Staubli VAL3: readText.dtx

public bool bBYPASS
public bool bCycle
public bool bCycleEnd = true
bool bGetSpeed = true
bool bMatlab
bool bReadEnd = true
bool bReadWait
public bool bResumeCycle
bool bTxtHeadOk
public bool bWriteEnd = true
frame fPrdFrame = {x=1610.363, y=33.376, z=-220.436, rx=-0.03, ry=0.18, rz=-39.644, fatherId=world[0]}
jointRx jJointRead[100]
  [0] = {j1=8.22, j2=20.1, j3=107.19, j4=-141.77, j5=44.38, j6=150.9}
  [1] = {j1=8.22, j2=20.1, j3=107.19, j4=-141.77, j5=44.38, j6=150.9}
public jointRx jPrdHome = {j1=40.635, j2=24.616, j3=104.715, j4=-108.663, j5=68.526, j6=132.709}
mdesc mNomSpeed = {accel=16, vel=40, decel=16, tmax=80, blend=off, leave=20, reach=20}
public mdesc mSpdOfJnt[100]
  [0] = {accel=40, vel=40, decel=40, rmax=1000, tmax=40, blend=cartesian, leave=0, reach=2}
  [1] = {accel=40, vel=40, decel=40, rmax=1000, tmax=40, blend=cartesian, leave=0, reach=2}
  [2] = {accel=30, vel=40, decel=30, rmax=1000, tmax=15.702, blend=cartesian, leave=0, reach=2}
  [3] = {accel=30, vel=40, decel=30, rmax=1000, tmax=6.112, blend=cartesian, leave=0, reach=2}
  [4] = {accel=16, vel=40, decel=16, rmax=1000, tmax=200, blend=cartesian, leave=2, reach=2}
  [5] = {accel=16, vel=40, decel=16, rmax=1000, tmax=200, blend=cartesian, leave=2, reach=2}
  [6] = {accel=16, vel=40, decel=16, rmax=1000, tmax=200, blend=cartesian, leave=2, reach=2}
  [7] = {accel=16, vel=40, decel=16, rmax=1000, tmax=200, blend=cartesian, leave=2, reach=2}
  [8] = {accel=16, vel=40, decel=16, rmax=1000, tmax=200, blend=cartesian, leave=2, reach=2}
  [9] = {accel=16, vel=40, decel=16, rmax=1000, tmax=200, blend=cartesian, leave=2, reach=2}
  [10] = {accel=16, vel=40, decel=16, rmax=1000, tmax=200, blend=cartesian, leave=2, reach=2}
  [11] = {accel=16, vel=40, decel=16, rmax=1000, tmax=200, blend=cartesian, leave=2, reach=2}
  [12] = {accel=16, vel=40, decel=16, rmax=1000, tmax=200, blend=cartesian, leave=2, reach=2}
  [13] = {accel=16, vel=40, decel=16, rmax=1000, tmax=200, blend=cartesian, leave=2, reach=2}
  [14] = {accel=16, vel=40, decel=16, rmax=1000, tmax=200, blend=cartesian, leave=2, reach=2}
  [15] = {accel=16, vel=40, decel=16, rmax=1000, tmax=200, blend=cartesian, leave=2, reach=2}
  [16] = {accel=16, vel=40, decel=16, rmax=1000, tmax=200, blend=cartesian, leave=2, reach=2}
  [17] = {accel=16, vel=40, decel=16, rmax=1000, tmax=200, blend=cartesian, leave=2, reach=2}
  [18] = {accel=16, vel=40, decel=16, rmax=1000, tmax=200, blend=cartesian, leave=2, reach=2}
  [19] = {accel=16, vel=40, decel=16, rmax=1000, tmax=200, blend=cartesian, leave=2, reach=2}
  [20] = {accel=16, vel=40, decel=16, rmax=1000, tmax=200, blend=cartesian, leave=2, reach=2}
  [21] = {accel=16, vel=40, decel=16, rmax=1000, tmax=200, blend=cartesian, leave=2, reach=2}
  [22] = {accel=16, vel=40, decel=16, rmax=1000, tmax=200, blend=cartesian, leave=2, reach=2}
  [23] = {accel=16, vel=40, decel=16, rmax=1000, tmax=200, blend=cartesian, leave=2, reach=2}
  [24] = {accel=16, vel=40, decel=16, rmax=1000, tmax=200, blend=cartesian, leave=2, reach=2}
  [25] = {accel=16, vel=40, decel=16, rmax=1000, tmax=200, blend=cartesian, leave=2, reach=2}
  [26] = {accel=16, vel=40, decel=16, rmax=1000, tmax=200, blend=cartesian, leave=2, reach=2}
  [27] = {accel=16, vel=40, decel=16, rmax=1000, tmax=200, blend=cartesian, leave=2, reach=2}
  [28] = {accel=16, vel=40, decel=16, rmax=1000, tmax=200, blend=cartesian, leave=2, reach=2}
  [29] = {accel=16, vel=40, decel=16, rmax=1000, tmax=200, blend=cartesian, leave=2, reach=2}
  [30] = {accel=16, vel=40, decel=16, rmax=1000, tmax=200, blend=cartesian, leave=2, reach=2}
  [31] = {accel=16, vel=40, decel=16, rmax=1000, tmax=200, blend=cartesian, leave=2, reach=2}
  [32] = {accel=16, vel=40, decel=16, rmax=1000, tmax=200, blend=cartesian, leave=2, reach=2}
  [33] = {accel=16, vel=40, decel=16, rmax=1000, tmax=200, blend=cartesian, leave=2, reach=2}
  [34] = {accel=16, vel=40, decel=16, rmax=1000, tmax=200, blend=cartesian, leave=2, reach=2}
  [35] = {accel=16, vel=40, decel=16, rmax=1000, tmax=200, blend=cartesian, leave=2, reach=2}
  [36] = {accel=16, vel=40, decel=16, rmax=1000, tmax=200, blend=cartesian, leave=2, reach=2}
  [37] = {accel=16, vel=40, decel=16, rmax=1000, tmax=200, blend=cartesian, leave=2, reach=2}
  [38] = {accel=16, vel=40, decel=16, rmax=1000, tmax=200, blend=cartesian, leave=2, reach=2}
  [39] = {accel=16, vel=40, decel=16, rmax=1000, tmax=200, blend=cartesian, leave=2, reach=2}
  [40] = {accel=16, vel=40, decel=16, rmax=1000, tmax=200, blend=cartesian, leave=2, reach=2}
  [41] = {accel=16, vel=40, decel=16, rmax=1000, tmax=200, blend=cartesian, leave=2, reach=2}
  [42] = {accel=16, vel=40, decel=16, rmax=1000, tmax=200, blend=cartesian, leave=2, reach=2}
  [43] = {accel=16, vel=40, decel=16, rmax=1000, tmax=200, blend=cartesian, leave=2, reach=2}
  [44] = {accel=16, vel=40, decel=16, rmax=1000, tmax=200, blend=cartesian, leave=2, reach=2}
  [45] = {accel=16, vel=40, decel=16, rmax=1000, tmax=200, blend=cartesian, leave=2, reach=2}
  [46] = {accel=16, vel=40, decel=16, rmax=1000, tmax=200, blend=cartesian, leave=2, reach=2}
  [47] = {accel=16, vel=40, decel=16, rmax=1000, tmax=200, blend=cartesian, leave=2, reach=2}
  [48] = {accel=16, vel=40, decel=16, rmax=1000, tmax=200, blend=cartesian, leave=2, reach=2}
  [49] = {accel=16, vel=40, decel=16, rmax=1000, tmax=200, blend=cartesian, leave=2, reach=2}
  [50] = {accel=16, vel=40, decel=16, rmax=1000, tmax=200, blend=cartesian, leave=2, reach=2}
  [51] = {accel=16, vel=40, decel=16, rmax=1000, tmax=200, blend=cartesian, leave=2, reach=2}
  [52] = {accel=16, vel=40, decel=16, rmax=1000, tmax=200, blend=cartesian, leave=2, reach=2}
  [53] = {accel=16, vel=40, decel=16, rmax=1000, tmax=200, blend=cartesian, leave=2, reach=2}
  [54] = {accel=16, vel=40, decel=16, rmax=1000, tmax=200, blend=cartesian, leave=2, reach=2}
  [55] = {accel=16, vel=40, decel=16, rmax=1000, tmax=200, blend=cartesian, leave=2, reach=2}
  [56] = {accel=16, vel=40, decel=16, rmax=1000, tmax=200, blend=cartesian, leave=2, reach=2}
  [57] = {accel=16, vel=40, decel=16, rmax=1000, tmax=200, blend=cartesian, leave=2, reach=2}
  [58] = {accel=16, vel=40, decel=16, rmax=1000, tmax=200, blend=cartesian, leave=2, reach=2}
  [59] = {accel=16, vel=40, decel=16, rmax=1000, tmax=200, blend=cartesian, leave=2, reach=2}
  [60] = {accel=16, vel=40, decel=16, rmax=1000, tmax=200, blend=cartesian, leave=2, reach=2}
  [61] = {accel=16, vel=40, decel=16, rmax=1000, tmax=200, blend=cartesian, leave=2, reach=2}
  [62] = {accel=16, vel=40, decel=16, rmax=1000, tmax=200, blend=cartesian, leave=2, reach=2}
  [63] = {accel=16, vel=40, decel=16, rmax=1000, tmax=200, blend=cartesian, leave=2, reach=2}
  [64] = {accel=16, vel=40, decel=16, rmax=1000, tmax=200, blend=cartesian, leave=2, reach=2}
  [65] = {accel=16, vel=40, decel=16, rmax=1000, tmax=200, blend=cartesian, leave=2, reach=2}
  [66] = {accel=16, vel=40, decel=16, rmax=1000, tmax=200, blend=cartesian, leave=2, reach=2}
  [67] = {accel=16, vel=40, decel=16, rmax=1000, tmax=200, blend=cartesian, leave=2, reach=2}
  [68] = {accel=16, vel=40, decel=16, rmax=1000, tmax=200, blend=cartesian, leave=2, reach=2}
  [69] = {accel=16, vel=40, decel=16, rmax=1000, tmax=200, blend=cartesian, leave=2, reach=2}
  [70] = {accel=16, vel=40, decel=16, rmax=1000, tmax=200, blend=cartesian, leave=2, reach=2}
  [71] = {accel=16, vel=40, decel=16, rmax=1000, tmax=200, blend=cartesian, leave=2, reach=2}
  [72] = {accel=16, vel=40, decel=16, rmax=1000, tmax=200, blend=cartesian, leave=2, reach=2}
  [73] = {accel=16, vel=40, decel=16, rmax=1000, tmax=200, blend=cartesian, leave=2, reach=2}
  [74] = {accel=16, vel=40, decel=16, rmax=1000, tmax=200, blend=cartesian, leave=2, reach=2}
  [75] = {accel=16, vel=40, decel=16, rmax=1000, tmax=200, blend=cartesian, leave=2, reach=2}
  [76] = {accel=16, vel=40, decel=16, rmax=1000, tmax=200, blend=cartesian, leave=2, reach=2}
  [77] = {accel=16, vel=40, decel=16, rmax=1000, tmax=200, blend=cartesian, leave=2, reach=2}
  [78] = {accel=16, vel=40, decel=16, rmax=1000, tmax=200, blend=cartesian, leave=2, reach=2}
  [79] = {accel=16, vel=40, decel=16, rmax=1000, tmax=200, blend=cartesian, leave=2, reach=2}
  [80] = {accel=16, vel=40, decel=16, rmax=1000, tmax=200, blend=cartesian, leave=2, reach=2}
  [81] = {accel=16, vel=40, decel=16, rmax=1000, tmax=200, blend=cartesian, leave=2, reach=2}
  [82] = {accel=16, vel=40, decel=16, rmax=1000, tmax=200, blend=cartesian, leave=2, reach=2}
  [83] = {accel=16, vel=40, decel=16, rmax=1000, tmax=200, blend=cartesian, leave=2, reach=2}
  [84] = {accel=16, vel=40, decel=16, rmax=1000, tmax=200, blend=cartesian, leave=2, reach=2}
  [85] = {accel=16, vel=40, decel=16, rmax=1000, tmax=200, blend=cartesian, leave=2, reach=2}
  [86] = {accel=16, vel=40, decel=16, rmax=1000, tmax=200, blend=cartesian, leave=2, reach=2}
  [87] = {accel=16, vel=40, decel=16, rmax=1000, tmax=200, blend=cartesian, leave=2, reach=2}
  [88] = {accel=16, vel=40, decel=16, rmax=1000, tmax=200, blend=cartesian, leave=2, reach=2}
  [89] = {accel=16, vel=40, decel=16, rmax=1000, tmax=200, blend=cartesian, leave=2, reach=2}
  [90] = {accel=16, vel=40, decel=16, rmax=1000, tmax=200, blend=cartesian, leave=2, reach=2}
  [91] = {accel=16, vel=40, decel=16, rmax=1000, tmax=200, blend=cartesian, leave=2, reach=2}
  [92] = {accel=16, vel=40, decel=16, rmax=1000, tmax=200, blend=cartesian, leave=2, reach=2}
  [93] = {accel=16, vel=40, decel=16, rmax=1000, tmax=200, blend=cartesian, leave=2, reach=2}
  [94] = {accel=16, vel=40, decel=16, rmax=1000, tmax=200, blend=cartesian, leave=2, reach=2}
  [95] = {accel=16, vel=40, decel=16, rmax=1000, tmax=200, blend=cartesian, leave=2, reach=2}
  [96] = {accel=16, vel=40, decel=16, rmax=1000, tmax=200, blend=cartesian, leave=2, reach=2}
  [97] = {accel=16, vel=40, decel=16, rmax=1000, tmax=200, blend=cartesian, leave=2, reach=2}
  [98] = {accel=16, vel=40, decel=16, rmax=1000, tmax=200, blend=cartesian, leave=2, reach=2}
  [99] = {accel=16, vel=40, decel=16, rmax=1000, tmax=200, blend=cartesian, leave=2, reach=2}
public mdesc mSpdOfPt[1000]
  [0] = {accel=80, decel=80, tmax=12.678, leave=0.5, reach=0.5}
  [1] = {accel=80, decel=80, tmax=11.985, leave=0.5, reach=0.5}
  [2] = {accel=80, decel=80, tmax=11.817, leave=0.5, reach=0.5}
  [3] = {accel=80, decel=80, tmax=11.196, leave=0.5, reach=0.5}
  [4] = {accel=80, decel=80, tmax=9.277, leave=0.5, reach=0.5}
  [5] = {accel=80, decel=80, tmax=7.453, leave=0.5, reach=0.5}
  [6] = {accel=80, decel=80, tmax=6.952, leave=0.5, reach=0.5}
  [7] = {accel=80, decel=80, tmax=7.802, leave=0.5, reach=0.5}
  [8] = {accel=80, decel=80, tmax=10.02, leave=0.5, reach=0.5}
  [9] = {accel=80, decel=80, tmax=12.345, leave=0.5, reach=0.5}
  [10] = {accel=80, decel=80, tmax=14.425, leave=0.5, reach=0.5}
  [11] = {accel=80, decel=80, tmax=15.256, leave=0.5, reach=0.5}
  [12] = {accel=80, decel=80, tmax=15.163, leave=0.5, reach=0.5}
  [13] = {accel=80, decel=80, tmax=13.825, leave=0.5, reach=0.5}
  [14] = {accel=80, decel=80, tmax=12.953, leave=0.5, reach=0.5}
  [15] = {accel=80, decel=80, tmax=11.37, leave=0.5, reach=0.5}
  [16] = {accel=80, decel=80, tmax=9.559, leave=0.5, reach=0.5}
  [17] = {accel=80, decel=80, tmax=9.004, leave=0.5, reach=0.5}
  [18] = {accel=80, decel=80, tmax=10.189, leave=0.5, reach=0.5}
  [19] = {accel=80, decel=80, tmax=12.733, leave=0.5, reach=0.5}
  [20] = {accel=80, decel=80, tmax=10.204, leave=0.5, reach=0.5}
  [21] = {accel=80, decel=80, tmax=6.338, leave=0.5, reach=0.5}
  [22] = {accel=80, decel=80, tmax=4.399, leave=0.5, reach=0.5}
  [23] = {accel=80, decel=80, tmax=3.23, leave=0.5, reach=0.5}
  [24] = {accel=80, decel=80, tmax=3.6, leave=0.5, reach=0.5}
  [25] = {accel=80, decel=80, tmax=5.733, leave=0.5, reach=0.5}
  [26] = {accel=80, decel=80, tmax=10.337, leave=0.5, reach=0.5}
  [27] = {accel=80, decel=80, tmax=12.442, leave=0.5, reach=0.5}
  [28] = {accel=80, decel=80, tmax=8.009, leave=0.5, reach=0.5}
  [29] = {accel=80, decel=80, tmax=7.489, leave=0.5, reach=0.5}
  [30] = {accel=80, decel=80, tmax=9.024, leave=0.5, reach=0.5}
  [31] = {accel=80, decel=80, tmax=10.72, leave=0.5, reach=0.5}
  [32] = {accel=80, decel=80, tmax=13.479, leave=0.5, reach=0.5}
  [33] = {accel=80, decel=80, tmax=15.007, leave=0.5, reach=0.5}
  [34] = {accel=80, decel=80, tmax=16.256, leave=0.5, reach=0.5}
  [35] = {accel=80, decel=80, tmax=14.52, leave=0.5, reach=0.5}
  [36] = {accel=80, decel=80, tmax=13.789, leave=0.5, reach=0.5}
  [37] = {accel=80, decel=80, tmax=13.032, leave=0.5, reach=0.5}
  [38] = {accel=80, decel=80, tmax=10.441, leave=0.5, reach=0.5}
  [39] = {accel=80, decel=80, tmax=8.528, leave=0.5, reach=0.5}
  [40] = {accel=80, decel=80, tmax=7.32, leave=0.5, reach=0.5}
  [41] = {accel=80, decel=80, tmax=7.727, leave=0.5, reach=0.5}
  [42] = {accel=80, decel=80, tmax=9.914, leave=0.5, reach=0.5}
  [43] = {accel=80, decel=80, tmax=12.183, leave=0.5, reach=0.5}
  [44] = {accel=80, decel=80, tmax=11.946, leave=0.5, reach=0.5}
  [45] = {accel=80, decel=80, tmax=11.661, leave=0.5, reach=0.5}
  [46] = {accel=80, decel=80, tmax=12.164, leave=0.5, reach=0.5}
  [47] = {accel=80, decel=80, tmax=13.305, leave=0.5, reach=0.5}
  [48] = {accel=80, decel=80, tmax=14.537, leave=0.5, reach=0.5}
  [49] = {accel=80, decel=80, tmax=14.655, leave=0.5, reach=0.5}
  [50] = {accel=80, decel=80, tmax=13.906, leave=0.5, reach=0.5}
  [51] = {accel=80, decel=80, tmax=12.405, leave=0.5, reach=0.5}
  [52] = {accel=80, decel=80, tmax=11.068, leave=0.5, reach=0.5}
  [53] = {accel=80, decel=80, tmax=9.816, leave=0.5, reach=0.5}
  [54] = {accel=80, decel=80, tmax=8.99, leave=0.5, reach=0.5}
  [55] = {accel=80, decel=80, tmax=8.736, leave=0.5, reach=0.5}
  [56] = {accel=80, decel=80, tmax=8.829, leave=0.5, reach=0.5}
  [57] = {accel=80, decel=80, tmax=9.678, leave=0.5, reach=0.5}
  [58] = {accel=80, decel=80, tmax=11.32, leave=0.5, reach=0.5}
  [59] = {accel=80, decel=80, tmax=13.047, leave=0.5, reach=0.5}
  [60] = {accel=80, decel=80, tmax=14.414, leave=0.5, reach=0.5}
  [61] = {accel=80, decel=80, tmax=14.8, leave=0.5, reach=0.5}
  [62] = {accel=80, decel=80, tmax=15.263, leave=0.5, reach=0.5}
  [63] = {accel=80, decel=80, tmax=15.263, leave=0.5, reach=0.5}
  [64] = {accel=80, decel=80, tmax=14.8, leave=0.5, reach=0.5}
  [65] = {accel=80, decel=80, tmax=14.414, leave=0.5, reach=0.5}
  [66] = {accel=80, decel=80, tmax=13.047, leave=0.5, reach=0.5}
  [67] = {accel=80, decel=80, tmax=11.32, leave=0.5, reach=0.5}
  [68] = {accel=80, decel=80, tmax=9.678, leave=0.5, reach=0.5}
  [69] = {accel=80, decel=80, tmax=8.829, leave=0.5, reach=0.5}
  [70] = {accel=80, decel=80, tmax=8.736, leave=0.5, reach=0.5}
  [71] = {accel=80, decel=80, tmax=8.99, leave=0.5, reach=0.5}
  [72] = {accel=80, decel=80, tmax=9.816, leave=0.5, reach=0.5}
  [73] = {accel=80, decel=80, tmax=11.068, leave=0.5, reach=0.5}
  [74] = {accel=80, decel=80, tmax=12.405, leave=0.5, reach=0.5}
  [75] = {accel=80, decel=80, tmax=13.906, leave=0.5, reach=0.5}
  [76] = {accel=80, decel=80, tmax=14.655, leave=0.5, reach=0.5}
  [77] = {accel=80, decel=80, tmax=14.537, leave=0.5, reach=0.5}
  [78] = {accel=80, decel=80, tmax=13.305, leave=0.5, reach=0.5}
  [79] = {accel=80, decel=80, tmax=12.164, leave=0.5, reach=0.5}
  [80] = {accel=80, decel=80, tmax=11.661, leave=0.5, reach=0.5}
  [81] = {accel=80, decel=80, tmax=11.946, leave=0.5, reach=0.5}
  [82] = {accel=80, decel=80, tmax=12.183, leave=0.5, reach=0.5}
  [83] = {accel=80, decel=80, tmax=9.914, leave=0.5, reach=0.5}
  [84] = {accel=80, decel=80, tmax=7.727, leave=0.5, reach=0.5}
  [85] = {accel=80, decel=80, tmax=7.32, leave=0.5, reach=0.5}
  [86] = {accel=80, decel=80, tmax=8.528, leave=0.5, reach=0.5}
  [87] = {accel=80, decel=80, tmax=10.441, leave=0.5, reach=0.5}
  [88] = {accel=80, decel=80, tmax=13.032, leave=0.5, reach=0.5}
  [89] = {accel=80, decel=80, tmax=13.789, leave=0.5, reach=0.5}
  [90] = {accel=80, decel=80, tmax=14.52, leave=0.5, reach=0.5}
  [91] = {accel=80, decel=80, tmax=16.256, leave=0.5, reach=0.5}
  [92] = {accel=80, decel=80, tmax=15.007, leave=0.5, reach=0.5}
  [93] = {accel=80, decel=80, tmax=13.479, leave=0.5, reach=0.5}
  [94] = {accel=80, decel=80, tmax=10.72, leave=0.5, reach=0.5}
  [95] = {accel=80, decel=80, tmax=9.024, leave=0.5, reach=0.5}
  [96] = {accel=80, decel=80, tmax=7.489, leave=0.5, reach=0.5}
  [97] = {accel=80, decel=80, tmax=8.009, leave=0.5, reach=0.5}
  [98] = {accel=80, decel=80, tmax=12.442, leave=0.5, reach=0.5}
  [99] = {accel=80, decel=80, tmax=10.337, leave=0.5, reach=0.5}
  [100] = {accel=80, decel=80, tmax=5.733, leave=0.5, reach=0.5}
  [101] = {accel=80, decel=80, tmax=3.6, leave=0.5, reach=0.5}
  [102] = {accel=80, decel=80, tmax=2.543, leave=0.5, reach=0.5}
  [103] = {accel=80, decel=80, tmax=3.382, leave=0.5, reach=0.5}
  [104] = {accel=80, decel=80, tmax=8.429, leave=0.5, reach=0.5}
  [105] = {accel=80, decel=80, tmax=19.886, leave=0.5, reach=0.5}
  [106] = {accel=80, decel=80, tmax=17.791, leave=0.5, reach=0.5}
  [107] = {accel=80, decel=80, tmax=11.419, leave=0.5, reach=0.5}
  [108] = {accel=80, decel=80, tmax=11.37, leave=0.5, reach=0.5}
  [109] = {accel=80, decel=80, tmax=11.627, leave=0.5, reach=0.5}
  [110] = {accel=80, decel=80, tmax=12.894, leave=0.5, reach=0.5}
  [111] = {accel=80, decel=80, tmax=13.668, leave=0.5, reach=0.5}
  [112] = {accel=80, decel=80, tmax=13.576, leave=0.5, reach=0.5}
  [113] = {accel=80, decel=80, tmax=14.175, leave=0.5, reach=0.5}
  [114] = {accel=80, decel=80, tmax=14.134, leave=0.5, reach=0.5}
  [115] = {accel=80, decel=80, tmax=13.985, leave=0.5, reach=0.5}
  [116] = {accel=80, decel=80, tmax=12.607, leave=0.5, reach=0.5}
  [117] = {accel=80, decel=80, tmax=11.516, leave=0.5, reach=0.5}
  [118] = {accel=80, decel=80, tmax=9.221, leave=0.5, reach=0.5}
  [119] = {accel=80, decel=80, tmax=7.688, leave=0.5, reach=0.5}
  [120] = {accel=80, decel=80, tmax=8.33, leave=0.5, reach=0.5}
  [121] = {accel=80, decel=80, tmax=12.323, leave=0.5, reach=0.5}
  [122] = {accel=80, decel=80, tmax=16.24, leave=0.5, reach=0.5}
  [123] = {accel=80, decel=80, tmax=16.452, leave=0.5, reach=0.5}
  [124] = {accel=80, decel=80, tmax=15.039, leave=0.5, reach=0.5}
  [125] = {accel=80, decel=80, tmax=15.151, leave=0.5, reach=0.5}
  [126] = {accel=80, decel=80, tmax=16.662, leave=0.5, reach=0.5}
  [127] = {accel=80, decel=80, tmax=17.112, leave=0.5, reach=0.5}
  [128] = {accel=80, decel=80, tmax=17.817, leave=0.5, reach=0.5}
  [129] = {accel=80, decel=80, tmax=16.855, leave=0.5, reach=0.5}
  [130] = {accel=80, decel=80, tmax=16.144, leave=0.5, reach=0.5}
  [131] = {accel=80, decel=80, tmax=13.939, leave=0.5, reach=0.5}
  [132] = {accel=80, decel=80, tmax=12.086, leave=0.5, reach=0.5}
  [133] = {accel=80, decel=80, tmax=11.201, leave=0.5, reach=0.5}
  [134] = {accel=80, decel=80, tmax=10.554, leave=0.5, reach=0.5}
  [135] = {accel=80, decel=80, tmax=10.969, leave=0.5, reach=0.5}
  [136] = {accel=80, decel=80, tmax=12.181, leave=0.5, reach=0.5}
  [137] = {accel=80, decel=80, tmax=14.738, leave=0.5, reach=0.5}
  [138] = {accel=80, decel=80, tmax=18.232, leave=0.5, reach=0.5}
  [139] = {accel=80, decel=80, tmax=21.108, leave=0.5, reach=0.5}
  [140] = {accel=80, decel=80, tmax=21.399, leave=0.5, reach=0.5}
  [141] = {accel=80, decel=80, tmax=21.285, leave=0.5, reach=0.5}
  [142] = {accel=80, decel=80, tmax=21.285, leave=0.5, reach=0.5}
  [143] = {accel=80, decel=80, tmax=21.399, leave=0.5, reach=0.5}
  [144] = {accel=80, decel=80, tmax=21.108, leave=0.5, reach=0.5}
  [145] = {accel=80, decel=80, tmax=18.232, leave=0.5, reach=0.5}
  [146] = {accel=80, decel=80, tmax=14.738, leave=0.5, reach=0.5}
  [147] = {accel=80, decel=80, tmax=12.181, leave=0.5, reach=0.5}
  [148] = {accel=80, decel=80, tmax=10.969, leave=0.5, reach=0.5}
  [149] = {accel=80, decel=80, tmax=10.554, leave=0.5, reach=0.5}
  [150] = {accel=80, decel=80, tmax=11.201, leave=0.5, reach=0.5}
  [151] = {accel=80, decel=80, tmax=12.086, leave=0.5, reach=0.5}
  [152] = {accel=80, decel=80, tmax=13.939, leave=0.5, reach=0.5}
  [153] = {accel=80, decel=80, tmax=16.144, leave=0.5, reach=0.5}
  [154] = {accel=80, decel=80, tmax=16.855, leave=0.5, reach=0.5}
  [155] = {accel=80, decel=80, tmax=17.817, leave=0.5, reach=0.5}
  [156] = {accel=80, decel=80, tmax=17.112, leave=0.5, reach=0.5}
  [157] = {accel=80, decel=80, tmax=16.662, leave=0.5, reach=0.5}
  [158] = {accel=80, decel=80, tmax=15.151, leave=0.5, reach=0.5}
  [159] = {accel=80, decel=80, tmax=15.039, leave=0.5, reach=0.5}
  [160] = {accel=80, decel=80, tmax=16.452, leave=0.5, reach=0.5}
  [161] = {accel=80, decel=80, tmax=16.24, leave=0.5, reach=0.5}
  [162] = {accel=80, decel=80, tmax=12.323, leave=0.5, reach=0.5}
  [163] = {accel=80, decel=80, tmax=8.33, leave=0.5, reach=0.5}
  [164] = {accel=80, decel=80, tmax=7.688, leave=0.5, reach=0.5}
  [165] = {accel=80, decel=80, tmax=9.221, leave=0.5, reach=0.5}
  [166] = {accel=80, decel=80, tmax=11.516, leave=0.5, reach=0.5}
  [167] = {accel=80, decel=80, tmax=12.607, leave=0.5, reach=0.5}
  [168] = {accel=80, decel=80, tmax=13.985, leave=0.5, reach=0.5}
  [169] = {accel=80, decel=80, tmax=14.134, leave=0.5, reach=0.5}
  [170] = {accel=80, decel=80, tmax=14.175, leave=0.5, reach=0.5}
  [171] = {accel=80, decel=80, tmax=13.576, leave=0.5, reach=0.5}
  [172] = {accel=80, decel=80, tmax=13.668, leave=0.5, reach=0.5}
  [173] = {accel=80, decel=80, tmax=12.894, leave=0.5, reach=0.5}
  [174] = {accel=80, decel=80, tmax=11.627, leave=0.5, reach=0.5}
  [175] = {accel=80, decel=80, tmax=11.37, leave=0.5, reach=0.5}
  [176] = {accel=80, decel=80, tmax=11.419, leave=0.5, reach=0.5}
  [177] = {accel=80, decel=80, tmax=17.791, leave=0.5, reach=0.5}
  [178] = {accel=80, decel=80, tmax=19.886, leave=0.5, reach=0.5}
  [179] = {accel=80, decel=80, tmax=8.429, leave=0.5, reach=0.5}
  [180] = {accel=80, decel=80, tmax=3.382, leave=0.5, reach=0.5}
  [181] = {accel=80, decel=80, tmax=2.528, leave=0.5, reach=0.5}
  [182] = {accel=80, decel=80, tmax=5.122, leave=0.5, reach=0.5}
  [183] = {accel=80, decel=80, tmax=27.24, leave=0.5, reach=0.5}
  [184] = {accel=80, decel=80, tmax=39.096, leave=0.5, reach=0.5}
  [185] = {accel=80, decel=80, tmax=33.981, leave=0.5, reach=0.5}
  [186] = {accel=80, decel=80, tmax=21.665, leave=0.5, reach=0.5}
  [187] = {accel=80, decel=80, tmax=15.615, leave=0.5, reach=0.5}
  [188] = {accel=80, decel=80, tmax=14.794, leave=0.5, reach=0.5}
  [189] = {accel=80, decel=80, tmax=14.111, leave=0.5, reach=0.5}
  [190] = {accel=80, decel=80, tmax=11.648, leave=0.5, reach=0.5}
  [191] = {accel=80, decel=80, tmax=10.193, leave=0.5, reach=0.5}
  [192] = {accel=80, decel=80, tmax=9.944, leave=0.5, reach=0.5}
  [193] = {accel=80, decel=80, tmax=9.415, leave=0.5, reach=0.5}
  [194] = {accel=80, decel=80, tmax=9.98, leave=0.5, reach=0.5}
  [195] = {accel=80, decel=80, tmax=10.948, leave=0.5, reach=0.5}
  [196] = {accel=80, decel=80, tmax=10.247, leave=0.5, reach=0.5}
  [197] = {accel=80, decel=80, tmax=9.066, leave=0.5, reach=0.5}
  [198] = {accel=80, decel=80, tmax=8.169, leave=0.5, reach=0.5}
  [199] = {accel=80, decel=80, tmax=9.444, leave=0.5, reach=0.5}
  [200] = {accel=80, decel=80, tmax=14.904, leave=0.5, reach=0.5}
  [201] = {accel=80, decel=80, tmax=23.746, leave=0.5, reach=0.5}
  [202] = {accel=80, decel=80, tmax=21.93, leave=0.5, reach=0.5}
  [203] = {accel=80, decel=80, tmax=18.32, leave=0.5, reach=0.5}
  [204] = {accel=80, decel=80, tmax=18.189, leave=0.5, reach=0.5}
  [205] = {accel=80, decel=80, tmax=16.627, leave=0.5, reach=0.5}
  [206] = {accel=80, decel=80, tmax=16.144, leave=0.5, reach=0.5}
  [207] = {accel=80, decel=80, tmax=15.272, leave=0.5, reach=0.5}
  [208] = {accel=80, decel=80, tmax=14.535, leave=0.5, reach=0.5}
  [209] = {accel=80, decel=80, tmax=13.64, leave=0.5, reach=0.5}
  [210] = {accel=80, decel=80, tmax=12.328, leave=0.5, reach=0.5}
  [211] = {accel=80, decel=80, tmax=11.644, leave=0.5, reach=0.5}
  [212] = {accel=80, decel=80, tmax=10.7, leave=0.5, reach=0.5}
  [213] = {accel=80, decel=80, tmax=10.628, leave=0.5, reach=0.5}
  [214] = {accel=80, decel=80, tmax=10.811, leave=0.5, reach=0.5}
  [215] = {accel=80, decel=80, tmax=11.389, leave=0.5, reach=0.5}
  [216] = {accel=80, decel=80, tmax=13.021, leave=0.5, reach=0.5}
  [217] = {accel=80, decel=80, tmax=14.932, leave=0.5, reach=0.5}
  [218] = {accel=80, decel=80, tmax=15.176, leave=0.5, reach=0.5}
  [219] = {accel=80, decel=80, tmax=14.927, leave=0.5, reach=0.5}
  [220] = {accel=80, decel=80, tmax=14.802, leave=0.5, reach=0.5}
  [221] = {accel=80, decel=80, tmax=14.802, leave=0.5, reach=0.5}
  [222] = {accel=80, decel=80, tmax=14.927, leave=0.5, reach=0.5}
  [223] = {accel=80, decel=80, tmax=15.176, leave=0.5, reach=0.5}
  [224] = {accel=80, decel=80, tmax=14.932, leave=0.5, reach=0.5}
  [225] = {accel=80, decel=80, tmax=13.021, leave=0.5, reach=0.5}
  [226] = {accel=80, decel=80, tmax=11.389, leave=0.5, reach=0.5}
  [227] = {accel=80, decel=80, tmax=10.811, leave=0.5, reach=0.5}
  [228] = {accel=80, decel=80, tmax=10.628, leave=0.5, reach=0.5}
  [229] = {accel=80, decel=80, tmax=10.7, leave=0.5, reach=0.5}
  [230] = {accel=80, decel=80, tmax=11.644, leave=0.5, reach=0.5}
  [231] = {accel=80, decel=80, tmax=12.328, leave=0.5, reach=0.5}
  [232] = {accel=80, decel=80, tmax=13.64, leave=0.5, reach=0.5}
  [233] = {accel=80, decel=80, tmax=14.535, leave=0.5, reach=0.5}
  [234] = {accel=80, decel=80, tmax=15.272, leave=0.5, reach=0.5}
  [235] = {accel=80, decel=80, tmax=16.144, leave=0.5, reach=0.5}
  [236] = {accel=80, decel=80, tmax=16.627, leave=0.5, reach=0.5}
  [237] = {accel=80, decel=80, tmax=18.189, leave=0.5, reach=0.5}
  [238] = {accel=80, decel=80, tmax=18.32, leave=0.5, reach=0.5}
  [239] = {accel=80, decel=80, tmax=21.93, leave=0.5, reach=0.5}
  [240] = {accel=80, decel=80, tmax=23.746, leave=0.5, reach=0.5}
  [241] = {accel=80, decel=80, tmax=14.904, leave=0.5, reach=0.5}
  [242] = {accel=80, decel=80, tmax=9.444, leave=0.5, reach=0.5}
  [243] = {accel=80, decel=80, tmax=8.169, leave=0.5, reach=0.5}
  [244] = {accel=80, decel=80, tmax=9.066, leave=0.5, reach=0.5}
  [245] = {accel=80, decel=80, tmax=10.247, leave=0.5, reach=0.5}
  [246] = {accel=80, decel=80, tmax=10.948, leave=0.5, reach=0.5}
  [247] = {accel=80, decel=80, tmax=9.98, leave=0.5, reach=0.5}
  [248] = {accel=80, decel=80, tmax=9.415, leave=0.5, reach=0.5}
  [249] = {accel=80, decel=80, tmax=9.944, leave=0.5, reach=0.5}
  [250] = {accel=80, decel=80, tmax=10.193, leave=0.5, reach=0.5}
  [251] = {accel=80, decel=80, tmax=11.648, leave=0.5, reach=0.5}
  [252] = {accel=80, decel=80, tmax=14.111, leave=0.5, reach=0.5}
  [253] = {accel=80, decel=80, tmax=14.794, leave=0.5, reach=0.5}
  [254] = {accel=80, decel=80, tmax=15.615, leave=0.5, reach=0.5}
  [255] = {accel=80, decel=80, tmax=21.665, leave=0.5, reach=0.5}
  [256] = {accel=80, decel=80, tmax=33.981, leave=0.5, reach=0.5}
  [257] = {accel=80, decel=80, tmax=39.096, leave=0.5, reach=0.5}
  [258] = {accel=80, decel=80, tmax=27.24, leave=0.5, reach=0.5}
  [259] = {accel=80, decel=80, tmax=5.122, leave=0.5, reach=0.5}
  [260] = {accel=80, decel=80, tmax=2.547, leave=0.5, reach=0.5}
  [261] = {accel=80, decel=80, tmax=3.681, leave=0.5, reach=0.5}
  [262] = {accel=80, decel=80, tmax=13.149, leave=0.5, reach=0.5}
  [263] = {accel=80, decel=80, tmax=39.1, leave=0.5, reach=0.5}
  [264] = {accel=80, decel=80, tmax=22.809, leave=0.5, reach=0.5}
  [265] = {accel=80, decel=80, tmax=10.899, leave=0.5, reach=0.5}
  [266] = {accel=80, decel=80, tmax=8.399, leave=0.5, reach=0.5}
  [267] = {accel=80, decel=80, tmax=8.167, leave=0.5, reach=0.5}
  [268] = {accel=80, decel=80, tmax=7.52, leave=0.5, reach=0.5}
  [269] = {accel=80, decel=80, tmax=7.268, leave=0.5, reach=0.5}
  [270] = {accel=80, decel=80, tmax=7.004, leave=0.5, reach=0.5}
  [271] = {accel=80, decel=80, tmax=7.184, leave=0.5, reach=0.5}
  [272] = {accel=80, decel=80, tmax=7.999, leave=0.5, reach=0.5}
  [273] = {accel=80, decel=80, tmax=8.571, leave=0.5, reach=0.5}
  [274] = {accel=80, decel=80, tmax=8.981, leave=0.5, reach=0.5}
  [275] = {accel=80, decel=80, tmax=8.329, leave=0.5, reach=0.5}
  [276] = {accel=80, decel=80, tmax=7.046, leave=0.5, reach=0.5}
  [277] = {accel=80, decel=80, tmax=6.123, leave=0.5, reach=0.5}
  [278] = {accel=80, decel=80, tmax=6.509, leave=0.5, reach=0.5}
  [279] = {accel=80, decel=80, tmax=8.855, leave=0.5, reach=0.5}
  [280] = {accel=80, decel=80, tmax=10.441, leave=0.5, reach=0.5}
  [281] = {accel=80, decel=80, tmax=9.991, leave=0.5, reach=0.5}
  [282] = {accel=80, decel=80, tmax=9.233, leave=0.5, reach=0.5}
  [283] = {accel=80, decel=80, tmax=9.606, leave=0.5, reach=0.5}
  [284] = {accel=80, decel=80, tmax=9.957, leave=0.5, reach=0.5}
  [285] = {accel=80, decel=80, tmax=9.852, leave=0.5, reach=0.5}
  [286] = {accel=80, decel=80, tmax=9.886, leave=0.5, reach=0.5}
  [287] = {accel=80, decel=80, tmax=8.922, leave=0.5, reach=0.5}
  [288] = {accel=80, decel=80, tmax=8.344, leave=0.5, reach=0.5}
  [289] = {accel=80, decel=80, tmax=7.852, leave=0.5, reach=0.5}
  [290] = {accel=80, decel=80, tmax=7.47, leave=0.5, reach=0.5}
  [291] = {accel=80, decel=80, tmax=7.248, leave=0.5, reach=0.5}
  [292] = {accel=80, decel=80, tmax=6.848, leave=0.5, reach=0.5}
  [293] = {accel=80, decel=80, tmax=6.788, leave=0.5, reach=0.5}
  [294] = {accel=80, decel=80, tmax=7.003, leave=0.5, reach=0.5}
  [295] = {accel=80, decel=80, tmax=7.444, leave=0.5, reach=0.5}
  [296] = {accel=80, decel=80, tmax=8.022, leave=0.5, reach=0.5}
  [297] = {accel=80, decel=80, tmax=8.343, leave=0.5, reach=0.5}
  [298] = {accel=80, decel=80, tmax=8.488, leave=0.5, reach=0.5}
  [299] = {accel=80, decel=80, tmax=8.391, leave=0.5, reach=0.5}
  [300] = {accel=80, decel=80, tmax=8.391, leave=0.5, reach=0.5}
  [301] = {accel=80, decel=80, tmax=8.488, leave=0.5, reach=0.5}
  [302] = {accel=80, decel=80, tmax=8.343, leave=0.5, reach=0.5}
  [303] = {accel=80, decel=80, tmax=8.022, leave=0.5, reach=0.5}
  [304] = {accel=80, decel=80, tmax=7.444, leave=0.5, reach=0.5}
  [305] = {accel=80, decel=80, tmax=7.003, leave=0.5, reach=0.5}
  [306] = {accel=80, decel=80, tmax=6.788, leave=0.5, reach=0.5}
  [307] = {accel=80, decel=80, tmax=6.848, leave=0.5, reach=0.5}
  [308] = {accel=80, decel=80, tmax=7.248, leave=0.5, reach=0.5}
  [309] = {accel=80, decel=80, tmax=7.47, leave=0.5, reach=0.5}
  [310] = {accel=80, decel=80, tmax=7.852, leave=0.5, reach=0.5}
  [311] = {accel=80, decel=80, tmax=8.344, leave=0.5, reach=0.5}
  [312] = {accel=80, decel=80, tmax=8.922, leave=0.5, reach=0.5}
  [313] = {accel=80, decel=80, tmax=9.886, leave=0.5, reach=0.5}
  [314] = {accel=80, decel=80, tmax=9.852, leave=0.5, reach=0.5}
  [315] = {accel=80, decel=80, tmax=9.957, leave=0.5, reach=0.5}
  [316] = {accel=80, decel=80, tmax=9.606, leave=0.5, reach=0.5}
  [317] = {accel=80, decel=80, tmax=9.233, leave=0.5, reach=0.5}
  [318] = {accel=80, decel=80, tmax=9.991, leave=0.5, reach=0.5}
  [319] = {accel=80, decel=80, tmax=10.441, leave=0.5, reach=0.5}
  [320] = {accel=80, decel=80, tmax=8.855, leave=0.5, reach=0.5}
  [321] = {accel=80, decel=80, tmax=6.509, leave=0.5, reach=0.5}
  [322] = {accel=80, decel=80, tmax=6.123, leave=0.5, reach=0.5}
  [323] = {accel=80, decel=80, tmax=7.046, leave=0.5, reach=0.5}
  [324] = {accel=80, decel=80, tmax=8.329, leave=0.5, reach=0.5}
  [325] = {accel=80, decel=80, tmax=8.981, leave=0.5, reach=0.5}
  [326] = {accel=80, decel=80, tmax=8.571, leave=0.5, reach=0.5}
  [327] = {accel=80, decel=80, tmax=7.999, leave=0.5, reach=0.5}
  [328] = {accel=80, decel=80, tmax=7.184, leave=0.5, reach=0.5}
  [329] = {accel=80, decel=80, tmax=7.004, leave=0.5, reach=0.5}
  [330] = {accel=80, decel=80, tmax=7.268, leave=0.5, reach=0.5}
  [331] = {accel=80, decel=80, tmax=7.52, leave=0.5, reach=0.5}
  [332] = {accel=80, decel=80, tmax=8.167, leave=0.5, reach=0.5}
  [333] = {accel=80, decel=80, tmax=8.399, leave=0.5, reach=0.5}
  [334] = {accel=80, decel=80, tmax=10.899, leave=0.5, reach=0.5}
  [335] = {accel=80, decel=80, tmax=22.809, leave=0.5, reach=0.5}
  [336] = {accel=80, decel=80, tmax=39.1, leave=0.5, reach=0.5}
  [337] = {accel=80, decel=80, tmax=13.149, leave=0.5, reach=0.5}
  [338] = {accel=80, decel=80, tmax=3.681, leave=0.5, reach=0.5}
  [339] = {accel=80, decel=80, tmax=2.58, leave=0.5, reach=0.5}
  [340] = {accel=80, decel=80, tmax=3.155, leave=0.5, reach=0.5}
  [341] = {accel=80, decel=80, tmax=4.583, leave=0.5, reach=0.5}
  [342] = {accel=80, decel=80, tmax=10.995, leave=0.5, reach=0.5}
  [343] = {accel=80, decel=80, tmax=9.418, leave=0.5, reach=0.5}
  [344] = {accel=80, decel=80, tmax=5.253, leave=0.5, reach=0.5}
  [345] = {accel=80, decel=80, tmax=4.854, leave=0.5, reach=0.5}
  [346] = {accel=80, decel=80, tmax=5.307, leave=0.5, reach=0.5}
  [347] = {accel=80, decel=80, tmax=5.949, leave=0.5, reach=0.5}
  [348] = {accel=80, decel=80, tmax=7.318, leave=0.5, reach=0.5}
  [349] = {accel=80, decel=80, tmax=8.349, leave=0.5, reach=0.5}
  [350] = {accel=80, decel=80, tmax=8.382, leave=0.5, reach=0.5}
  [351] = {accel=80, decel=80, tmax=7.821, leave=0.5, reach=0.5}
  [352] = {accel=80, decel=80, tmax=6.717, leave=0.5, reach=0.5}
  [353] = {accel=80, decel=80, tmax=6.16, leave=0.5, reach=0.5}
  [354] = {accel=80, decel=80, tmax=5.083, leave=0.5, reach=0.5}
  [355] = {accel=80, decel=80, tmax=4.309, leave=0.5, reach=0.5}
  [356] = {accel=80, decel=80, tmax=3.973, leave=0.5, reach=0.5}
  [357] = {accel=80, decel=80, tmax=3.989, leave=0.5, reach=0.5}
  [358] = {accel=80, decel=80, tmax=4.577, leave=0.5, reach=0.5}
  [359] = {accel=80, decel=80, tmax=5.036, leave=0.5, reach=0.5}
  [360] = {accel=80, decel=80, tmax=5.057, leave=0.5, reach=0.5}
  [361] = {accel=80, decel=80, tmax=5.161, leave=0.5, reach=0.5}
  [362] = {accel=80, decel=80, tmax=5.668, leave=0.5, reach=0.5}
  [363] = {accel=80, decel=80, tmax=5.954, leave=0.5, reach=0.5}
  [364] = {accel=80, decel=80, tmax=6.248, leave=0.5, reach=0.5}
  [365] = {accel=80, decel=80, tmax=6.353, leave=0.5, reach=0.5}
  [366] = {accel=80, decel=80, tmax=6.079, leave=0.5, reach=0.5}
  [367] = {accel=80, decel=80, tmax=5.726, leave=0.5, reach=0.5}
  [368] = {accel=80, decel=80, tmax=5.206, leave=0.5, reach=0.5}
  [369] = {accel=80, decel=80, tmax=4.949, leave=0.5, reach=0.5}
  [370] = {accel=80, decel=80, tmax=4.649, leave=0.5, reach=0.5}
  [371] = {accel=80, decel=80, tmax=4.466, leave=0.5, reach=0.5}
  [372] = {accel=80, decel=80, tmax=4.472, leave=0.5, reach=0.5}
  [373] = {accel=80, decel=80, tmax=4.584, leave=0.5, reach=0.5}
  [374] = {accel=80, decel=80, tmax=4.826, leave=0.5, reach=0.5}
  [375] = {accel=80, decel=80, tmax=5.134, leave=0.5, reach=0.5}
  [376] = {accel=80, decel=80, tmax=5.318, leave=0.5, reach=0.5}
  [377] = {accel=80, decel=80, tmax=5.323, leave=0.5, reach=0.5}
  [378] = {accel=80, decel=80, tmax=5.318, leave=0.5, reach=0.5}
  [379] = {accel=80, decel=80, tmax=5.318, leave=0.5, reach=0.5}
  [380] = {accel=80, decel=80, tmax=5.323, leave=0.5, reach=0.5}
  [381] = {accel=80, decel=80, tmax=5.318, leave=0.5, reach=0.5}
  [382] = {accel=80, decel=80, tmax=5.134, leave=0.5, reach=0.5}
  [383] = {accel=80, decel=80, tmax=4.826, leave=0.5, reach=0.5}
  [384] = {accel=80, decel=80, tmax=4.584, leave=0.5, reach=0.5}
  [385] = {accel=80, decel=80, tmax=4.472, leave=0.5, reach=0.5}
  [386] = {accel=80, decel=80, tmax=4.466, leave=0.5, reach=0.5}
  [387] = {accel=80, decel=80, tmax=4.649, leave=0.5, reach=0.5}
  [388] = {accel=80, decel=80, tmax=4.949, leave=0.5, reach=0.5}
  [389] = {accel=80, decel=80, tmax=5.206, leave=0.5, reach=0.5}
  [390] = {accel=80, decel=80, tmax=5.726, leave=0.5, reach=0.5}
  [391] = {accel=80, decel=80, tmax=6.079, leave=0.5, reach=0.5}
  [392] = {accel=80, decel=80, tmax=6.353, leave=0.5, reach=0.5}
  [393] = {accel=80, decel=80, tmax=6.248, leave=0.5, reach=0.5}
  [394] = {accel=80, decel=80, tmax=5.954, leave=0.5, reach=0.5}
  [395] = {accel=80, decel=80, tmax=5.668, leave=0.5, reach=0.5}
  [396] = {accel=80, decel=80, tmax=5.161, leave=0.5, reach=0.5}
  [397] = {accel=80, decel=80, tmax=5.057, leave=0.5, reach=0.5}
  [398] = {accel=80, decel=80, tmax=5.036, leave=0.5, reach=0.5}
  [399] = {accel=80, decel=80, tmax=4.577, leave=0.5, reach=0.5}
  [400] = {accel=80, decel=80, tmax=3.989, leave=0.5, reach=0.5}
  [401] = {accel=80, decel=80, tmax=3.973, leave=0.5, reach=0.5}
  [402] = {accel=80, decel=80, tmax=4.309, leave=0.5, reach=0.5}
  [403] = {accel=80, decel=80, tmax=5.083, leave=0.5, reach=0.5}
  [404] = {accel=80, decel=80, tmax=6.16, leave=0.5, reach=0.5}
  [405] = {accel=80, decel=80, tmax=6.717, leave=0.5, reach=0.5}
  [406] = {accel=80, decel=80, tmax=7.821, leave=0.5, reach=0.5}
  [407] = {accel=80, decel=80, tmax=8.382, leave=0.5, reach=0.5}
  [408] = {accel=80, decel=80, tmax=8.349, leave=0.5, reach=0.5}
  [409] = {accel=80, decel=80, tmax=7.318, leave=0.5, reach=0.5}
  [410] = {accel=80, decel=80, tmax=5.949, leave=0.5, reach=0.5}
  [411] = {accel=80, decel=80, tmax=5.307, leave=0.5, reach=0.5}
  [412] = {accel=80, decel=80, tmax=4.854, leave=0.5, reach=0.5}
  [413] = {accel=80, decel=80, tmax=5.253, leave=0.5, reach=0.5}
  [414] = {accel=80, decel=80, tmax=9.418, leave=0.5, reach=0.5}
  [415] = {accel=80, decel=80, tmax=10.995, leave=0.5, reach=0.5}
  [416] = {accel=80, decel=80, tmax=4.583, leave=0.5, reach=0.5}
  [417] = {accel=80, decel=80, tmax=3.155, leave=0.5, reach=0.5}
  [418] = {accel=80, decel=80, tmax=3.258, leave=0.5, reach=0.5}
  [419] = {accel=80, decel=80, tmax=3.356, leave=0.5, reach=0.5}
  [420] = {accel=80, decel=80, tmax=2.648, leave=0.5, reach=0.5}
  [421] = {accel=80, decel=80, tmax=2.613, leave=0.5, reach=0.5}
  [422] = {accel=80, decel=80, tmax=2.6, leave=0.5, reach=0.5}
  [423] = {accel=80, decel=80, tmax=2.593, leave=0.5, reach=0.5}
  [424] = {accel=80, decel=80, tmax=3.227, leave=0.5, reach=0.5}
  [425] = {accel=80, decel=80, tmax=4.931, leave=0.5, reach=0.5}
  [426] = {accel=80, decel=80, tmax=7.775, leave=0.5, reach=0.5}
  [427] = {accel=80, decel=80, tmax=11.334, leave=0.5, reach=0.5}
  [428] = {accel=80, decel=80, tmax=15.093, leave=0.5, reach=0.5}
  [429] = {accel=80, decel=80, tmax=15.479, leave=0.5, reach=0.5}
  [430] = {accel=80, decel=80, tmax=13.175, leave=0.5, reach=0.5}
  [431] = {accel=80, decel=80, tmax=7.77, leave=0.5, reach=0.5}
  [432] = {accel=80, decel=80, tmax=5.6, leave=0.5, reach=0.5}
  [433] = {accel=80, decel=80, tmax=4.07, leave=0.5, reach=0.5}
  [434] = {accel=80, decel=80, tmax=3.359, leave=0.5, reach=0.5}
  [435] = {accel=80, decel=80, tmax=3.106, leave=0.5, reach=0.5}
  [436] = {accel=80, decel=80, tmax=3.155, leave=0.5, reach=0.5}
  [437] = {accel=80, decel=80, tmax=3.561, leave=0.5, reach=0.5}
  [438] = {accel=80, decel=80, tmax=3.68, leave=0.5, reach=0.5}
  [439] = {accel=80, decel=80, tmax=3.763, leave=0.5, reach=0.5}
  [440] = {accel=80, decel=80, tmax=3.989, leave=0.5, reach=0.5}
  [441] = {accel=80, decel=80, tmax=4.407, leave=0.5, reach=0.5}
  [442] = {accel=80, decel=80, tmax=4.962, leave=0.5, reach=0.5}
  [443] = {accel=80, decel=80, tmax=5.407, leave=0.5, reach=0.5}
  [444] = {accel=80, decel=80, tmax=5.814, leave=0.5, reach=0.5}
  [445] = {accel=80, decel=80, tmax=5.621, leave=0.5, reach=0.5}
  [446] = {accel=80, decel=80, tmax=5.29, leave=0.5, reach=0.5}
  [447] = {accel=80, decel=80, tmax=4.76, leave=0.5, reach=0.5}
  [448] = {accel=80, decel=80, tmax=4.196, leave=0.5, reach=0.5}
  [449] = {accel=80, decel=80, tmax=3.895, leave=0.5, reach=0.5}
  [450] = {accel=80, decel=80, tmax=3.762, leave=0.5, reach=0.5}
  [451] = {accel=80, decel=80, tmax=3.809, leave=0.5, reach=0.5}
  [452] = {accel=80, decel=80, tmax=3.939, leave=0.5, reach=0.5}
  [453] = {accel=80, decel=80, tmax=4.177, leave=0.5, reach=0.5}
  [454] = {accel=80, decel=80, tmax=4.497, leave=0.5, reach=0.5}
  [455] = {accel=80, decel=80, tmax=4.715, leave=0.5, reach=0.5}
  [456] = {accel=80, decel=80, tmax=4.875, leave=0.5, reach=0.5}
  [457] = {accel=80, decel=80, tmax=4.986, leave=0.5, reach=0.5}
  [458] = {accel=80, decel=80, tmax=4.986, leave=0.5, reach=0.5}
  [459] = {accel=80, decel=80, tmax=4.875, leave=0.5, reach=0.5}
  [460] = {accel=80, decel=80, tmax=4.715, leave=0.5, reach=0.5}
  [461] = {accel=80, decel=80, tmax=4.497, leave=0.5, reach=0.5}
  [462] = {accel=80, decel=80, tmax=4.177, leave=0.5, reach=0.5}
  [463] = {accel=80, decel=80, tmax=3.939, leave=0.5, reach=0.5}
  [464] = {accel=80, decel=80, tmax=3.809, leave=0.5, reach=0.5}
  [465] = {accel=80, decel=80, tmax=3.762, leave=0.5, reach=0.5}
  [466] = {accel=80, decel=80, tmax=3.895, leave=0.5, reach=0.5}
  [467] = {accel=80, decel=80, tmax=4.196, leave=0.5, reach=0.5}
  [468] = {accel=80, decel=80, tmax=4.76, leave=0.5, reach=0.5}
  [469] = {accel=80, decel=80, tmax=5.29, leave=0.5, reach=0.5}
  [470] = {accel=80, decel=80, tmax=5.621, leave=0.5, reach=0.5}
  [471] = {accel=80, decel=80, tmax=5.814, leave=0.5, reach=0.5}
  [472] = {accel=80, decel=80, tmax=5.407, leave=0.5, reach=0.5}
  [473] = {accel=80, decel=80, tmax=4.962, leave=0.5, reach=0.5}
  [474] = {accel=80, decel=80, tmax=4.407, leave=0.5, reach=0.5}
  [475] = {accel=80, decel=80, tmax=3.989, leave=0.5, reach=0.5}
  [476] = {accel=80, decel=80, tmax=3.763, leave=0.5, reach=0.5}
  [477] = {accel=80, decel=80, tmax=3.68, leave=0.5, reach=0.5}
  [478] = {accel=80, decel=80, tmax=3.561, leave=0.5, reach=0.5}
  [479] = {accel=80, decel=80, tmax=3.155, leave=0.5, reach=0.5}
  [480] = {accel=80, decel=80, tmax=3.106, leave=0.5, reach=0.5}
  [481] = {accel=80, decel=80, tmax=3.359, leave=0.5, reach=0.5}
  [482] = {accel=80, decel=80, tmax=4.07, leave=0.5, reach=0.5}
  [483] = {accel=80, decel=80, tmax=5.6, leave=0.5, reach=0.5}
  [484] = {accel=80, decel=80, tmax=7.77, leave=0.5, reach=0.5}
  [485] = {accel=80, decel=80, tmax=13.175, leave=0.5, reach=0.5}
  [486] = {accel=80, decel=80, tmax=15.479, leave=0.5, reach=0.5}
  [487] = {accel=80, decel=80, tmax=15.093, leave=0.5, reach=0.5}
  [488] = {accel=80, decel=80, tmax=11.334, leave=0.5, reach=0.5}
  [489] = {accel=80, decel=80, tmax=7.775, leave=0.5, reach=0.5}
  [490] = {accel=80, decel=80, tmax=4.931, leave=0.5, reach=0.5}
  [491] = {accel=80, decel=80, tmax=3.227, leave=0.5, reach=0.5}
  [492] = {accel=80, decel=80, tmax=2.593, leave=0.5, reach=0.5}
  [493] = {accel=80, decel=80, tmax=2.6, leave=0.5, reach=0.5}
  [494] = {accel=80, decel=80, tmax=2.613, leave=0.5, reach=0.5}
  [495] = {accel=80, decel=80, tmax=2.648, leave=0.5, reach=0.5}
  [496] = {accel=80, decel=80, tmax=2.333, leave=0.5, reach=0.5}
  [497] = {accel=80, decel=80, tmax=40, leave=0.5, reach=0.5}
  [498] = {accel=80, decel=80, tmax=12.235, leave=0.5, reach=0.5}
  [499] = {accel=80, decel=80, tmax=10.295, leave=0.5, reach=0.5}
  [500] = {accel=80, decel=80, tmax=8.845, leave=0.5, reach=0.5}
  [501] = {accel=80, decel=80, tmax=8.045, leave=0.5, reach=0.5}
  [502] = {accel=80, decel=80, tmax=7.797, leave=0.5, reach=0.5}
  [503] = {accel=80, decel=80, tmax=8.313, leave=0.5, reach=0.5}
  [504] = {accel=80, decel=80, tmax=9.406, leave=0.5, reach=0.5}
  [505] = {accel=80, decel=80, tmax=11.036, leave=0.5, reach=0.5}
  [506] = {accel=80, decel=80, tmax=12.697, leave=0.5, reach=0.5}
  [507] = {accel=80, decel=80, tmax=14.111, leave=0.5, reach=0.5}
  [508] = {accel=80, decel=80, tmax=14.961, leave=0.5, reach=0.5}
  [509] = {accel=80, decel=80, tmax=15.543, leave=0.5, reach=0.5}
  [510] = {accel=80, decel=80, tmax=15.543, leave=0.5, reach=0.5}
  [511] = {accel=80, decel=80, tmax=14.961, leave=0.5, reach=0.5}
  [512] = {accel=80, decel=80, tmax=14.111, leave=0.5, reach=0.5}
  [513] = {accel=80, decel=80, tmax=12.697, leave=0.5, reach=0.5}
  [514] = {accel=80, decel=80, tmax=11.036, leave=0.5, reach=0.5}
  [515] = {accel=80, decel=80, tmax=9.406, leave=0.5, reach=0.5}
  [516] = {accel=80, decel=80, tmax=8.313, leave=0.5, reach=0.5}
  [517] = {accel=80, decel=80, tmax=7.797, leave=0.5, reach=0.5}
  [518] = {accel=80, decel=80, tmax=8.045, leave=0.5, reach=0.5}
  [519] = {accel=80, decel=80, tmax=8.845, leave=0.5, reach=0.5}
  [520] = {accel=80, decel=80, tmax=10.295, leave=0.5, reach=0.5}
  [521] = {accel=80, decel=80, tmax=12.235, leave=0.5, reach=0.5}
  [522] = {accel=80, decel=80, tmax=14.178, leave=0.5, reach=0.5}
  [523] = {accel=80, decel=80, tmax=16.031, leave=0.5, reach=0.5}
  [524] = {accel=80, decel=80, tmax=16.724, leave=0.5, reach=0.5}
  [525] = {accel=80, decel=80, tmax=17.043, leave=0.5, reach=0.5}
  [526] = {accel=80, decel=80, tmax=16.4, leave=0.5, reach=0.5}
  [527] = {accel=80, decel=80, tmax=15.194, leave=0.5, reach=0.5}
  [528] = {accel=80, decel=80, tmax=13.575, leave=0.5, reach=0.5}
  [529] = {accel=80, decel=80, tmax=12.281, leave=0.5, reach=0.5}
  [530] = {accel=80, decel=80, tmax=11.268, leave=0.5, reach=0.5}
  [531] = {accel=80, decel=80, tmax=9.763, leave=0.5, reach=0.5}
  [532] = {accel=80, decel=80, tmax=8.886, leave=0.5, reach=0.5}
  [533] = {accel=80, decel=80, tmax=8.439, leave=0.5, reach=0.5}
  [534] = {accel=80, decel=80, tmax=8.897, leave=0.5, reach=0.5}
  [535] = {accel=80, decel=80, tmax=10.012, leave=0.5, reach=0.5}
  [536] = {accel=80, decel=80, tmax=12.344, leave=0.5, reach=0.5}
  [537] = {accel=80, decel=80, tmax=15.786, leave=0.5, reach=0.5}
  [538] = {accel=80, decel=80, tmax=19.207, leave=0.5, reach=0.5}
  [539] = {accel=80, decel=80, tmax=22.424, leave=0.5, reach=0.5}
  [540] = {accel=80, decel=80, tmax=21.581, leave=0.5, reach=0.5}
  [541] = {accel=80, decel=80, tmax=19.198, leave=0.5, reach=0.5}
  [542] = {accel=80, decel=80, tmax=15.91, leave=0.5, reach=0.5}
  [543] = {accel=80, decel=80, tmax=13.389, leave=0.5, reach=0.5}
  [544] = {accel=80, decel=80, tmax=12.656, leave=0.5, reach=0.5}
  [545] = {accel=80, decel=80, tmax=9.701, leave=0.5, reach=0.5}
  [546] = {accel=80, decel=80, tmax=8.018, leave=0.5, reach=0.5}
  [547] = {accel=80, decel=80, tmax=7.917, leave=0.5, reach=0.5}
  [548] = {accel=80, decel=80, tmax=8.748, leave=0.5, reach=0.5}
  [549] = {accel=80, decel=80, tmax=13.284, leave=0.5, reach=0.5}
  [550] = {accel=80, decel=80, tmax=13.35, leave=0.5, reach=0.5}
  [551] = {accel=80, decel=80, tmax=8.675, leave=0.5, reach=0.5}
  [552] = {accel=80, decel=80, tmax=8.318, leave=0.5, reach=0.5}
  [553] = {accel=80, decel=80, tmax=10.03, leave=0.5, reach=0.5}
  [554] = {accel=80, decel=80, tmax=13.62, leave=0.5, reach=0.5}
  [555] = {accel=80, decel=80, tmax=15.303, leave=0.5, reach=0.5}
  [556] = {accel=80, decel=80, tmax=15.363, leave=0.5, reach=0.5}
  [557] = {accel=80, decel=80, tmax=18.616, leave=0.5, reach=0.5}
  [558] = {accel=80, decel=80, tmax=21.441, leave=0.5, reach=0.5}
  [559] = {accel=80, decel=80, tmax=24.57, leave=0.5, reach=0.5}
  [560] = {accel=80, decel=80, tmax=23.361, leave=0.5, reach=0.5}
  [561] = {accel=80, decel=80, tmax=18.767, leave=0.5, reach=0.5}
  [562] = {accel=80, decel=80, tmax=14.287, leave=0.5, reach=0.5}
  [563] = {accel=80, decel=80, tmax=10.593, leave=0.5, reach=0.5}
  [564] = {accel=80, decel=80, tmax=8.688, leave=0.5, reach=0.5}
  [565] = {accel=80, decel=80, tmax=8.295, leave=0.5, reach=0.5}
  [566] = {accel=80, decel=80, tmax=8.977, leave=0.5, reach=0.5}
  [567] = {accel=80, decel=80, tmax=10.114, leave=0.5, reach=0.5}
  [568] = {accel=80, decel=80, tmax=11.529, leave=0.5, reach=0.5}
  [569] = {accel=80, decel=80, tmax=12.734, leave=0.5, reach=0.5}
  [570] = {accel=80, decel=80, tmax=14.354, leave=0.5, reach=0.5}
  [571] = {accel=80, decel=80, tmax=15.86, leave=0.5, reach=0.5}
  [572] = {accel=80, decel=80, tmax=17.094, leave=0.5, reach=0.5}
  [573] = {accel=80, decel=80, tmax=18.081, leave=0.5, reach=0.5}
  [574] = {accel=80, decel=80, tmax=19.235, leave=0.5, reach=0.5}
  [575] = {accel=80, decel=80, tmax=18.496, leave=0.5, reach=0.5}
  [576] = {accel=80, decel=80, tmax=16.121, leave=0.5, reach=0.5}
  [577] = {accel=80, decel=80, tmax=13.408, leave=0.5, reach=0.5}
  [578] = {accel=80, decel=80, tmax=10.765, leave=0.5, reach=0.5}
  [579] = {accel=80, decel=80, tmax=9.271, leave=0.5, reach=0.5}
  [580] = {accel=80, decel=80, tmax=8.168, leave=0.5, reach=0.5}
  [581] = {accel=80, decel=80, tmax=8.013, leave=0.5, reach=0.5}
  [582] = {accel=80, decel=80, tmax=8.598, leave=0.5, reach=0.5}
  [583] = {accel=80, decel=80, tmax=9.944, leave=0.5, reach=0.5}
  [584] = {accel=80, decel=80, tmax=11.822, leave=0.5, reach=0.5}
  [585] = {accel=80, decel=80, tmax=13.421, leave=0.5, reach=0.5}
  [586] = {accel=80, decel=80, tmax=14.72, leave=0.5, reach=0.5}
  [587] = {accel=80, decel=80, tmax=15.793, leave=0.5, reach=0.5}
  [588] = {accel=80, decel=80, tmax=16.515, leave=0.5, reach=0.5}
  [589] = {accel=80, decel=80, tmax=16.515, leave=0.5, reach=0.5}
  [590] = {accel=80, decel=80, tmax=15.793, leave=0.5, reach=0.5}
  [591] = {accel=80, decel=80, tmax=14.72, leave=0.5, reach=0.5}
  [592] = {accel=80, decel=80, tmax=13.421, leave=0.5, reach=0.5}
  [593] = {accel=80, decel=80, tmax=11.822, leave=0.5, reach=0.5}
  [594] = {accel=80, decel=80, tmax=9.944, leave=0.5, reach=0.5}
  [595] = {accel=80, decel=80, tmax=8.598, leave=0.5, reach=0.5}
  [596] = {accel=80, decel=80, tmax=8.013, leave=0.5, reach=0.5}
  [597] = {accel=80, decel=80, tmax=8.168, leave=0.5, reach=0.5}
  [598] = {accel=80, decel=80, tmax=9.271, leave=0.5, reach=0.5}
  [599] = {accel=80, decel=80, tmax=10.765, leave=0.5, reach=0.5}
  [600] = {accel=80, decel=80, tmax=13.408, leave=0.5, reach=0.5}
  [601] = {accel=80, decel=80, tmax=16.121, leave=0.5, reach=0.5}
  [602] = {accel=80, decel=80, tmax=18.496, leave=0.5, reach=0.5}
  [603] = {accel=80, decel=80, tmax=19.235, leave=0.5, reach=0.5}
  [604] = {accel=80, decel=80, tmax=18.081, leave=0.5, reach=0.5}
  [605] = {accel=80, decel=80, tmax=17.094, leave=0.5, reach=0.5}
  [606] = {accel=80, decel=80, tmax=15.86, leave=0.5, reach=0.5}
  [607] = {accel=80, decel=80, tmax=14.354, leave=0.5, reach=0.5}
  [608] = {accel=80, decel=80, tmax=12.734, leave=0.5, reach=0.5}
  [609] = {accel=80, decel=80, tmax=11.529, leave=0.5, reach=0.5}
  [610] = {accel=80, decel=80, tmax=10.114, leave=0.5, reach=0.5}
  [611] = {accel=80, decel=80, tmax=8.977, leave=0.5, reach=0.5}
  [612] = {accel=80, decel=80, tmax=8.295, leave=0.5, reach=0.5}
  [613] = {accel=80, decel=80, tmax=8.688, leave=0.5, reach=0.5}
  [614] = {accel=80, decel=80, tmax=10.593, leave=0.5, reach=0.5}
  [615] = {accel=80, decel=80, tmax=14.287, leave=0.5, reach=0.5}
  [616] = {accel=80, decel=80, tmax=18.767, leave=0.5, reach=0.5}
  [617] = {accel=80, decel=80, tmax=23.361, leave=0.5, reach=0.5}
  [618] = {accel=80, decel=80, tmax=24.57, leave=0.5, reach=0.5}
  [619] = {accel=80, decel=80, tmax=21.441, leave=0.5, reach=0.5}
  [620] = {accel=80, decel=80, tmax=18.616, leave=0.5, reach=0.5}
  [621] = {accel=80, decel=80, tmax=15.363, leave=0.5, reach=0.5}
  [622] = {accel=80, decel=80, tmax=15.303, leave=0.5, reach=0.5}
  [623] = {accel=80, decel=80, tmax=13.62, leave=0.5, reach=0.5}
  [624] = {accel=80, decel=80, tmax=10.03, leave=0.5, reach=0.5}
  [625] = {accel=80, decel=80, tmax=8.318, leave=0.5, reach=0.5}
  [626] = {accel=80, decel=80, tmax=8.675, leave=0.5, reach=0.5}
  [627] = {accel=80, decel=80, tmax=13.35, leave=0.5, reach=0.5}
  [628] = {accel=80, decel=80, tmax=14.902, leave=0.5, reach=0.5}
  [629] = {accel=80, decel=80, tmax=9.932, leave=0.5, reach=0.5}
  [630] = {accel=80, decel=80, tmax=7.277, leave=0.5, reach=0.5}
  [631] = {accel=80, decel=80, tmax=7.443, leave=0.5, reach=0.5}
  [632] = {accel=80, decel=80, tmax=10.629, leave=0.5, reach=0.5}
  [633] = {accel=80, decel=80, tmax=14.258, leave=0.5, reach=0.5}
  [634] = {accel=80, decel=80, tmax=14.257, leave=0.5, reach=0.5}
  [635] = {accel=80, decel=80, tmax=16.152, leave=0.5, reach=0.5}
  [636] = {accel=80, decel=80, tmax=20.378, leave=0.5, reach=0.5}
  [637] = {accel=80, decel=80, tmax=25.104, leave=0.5, reach=0.5}
  [638] = {accel=80, decel=80, tmax=28.756, leave=0.5, reach=0.5}
  [639] = {accel=80, decel=80, tmax=27.687, leave=0.5, reach=0.5}
  [640] = {accel=80, decel=80, tmax=24.489, leave=0.5, reach=0.5}
  [641] = {accel=80, decel=80, tmax=16.689, leave=0.5, reach=0.5}
  [642] = {accel=80, decel=80, tmax=12.173, leave=0.5, reach=0.5}
  [643] = {accel=80, decel=80, tmax=9.015, leave=0.5, reach=0.5}
  [644] = {accel=80, decel=80, tmax=7.904, leave=0.5, reach=0.5}
  [645] = {accel=80, decel=80, tmax=8.512, leave=0.5, reach=0.5}
  [646] = {accel=80, decel=80, tmax=9.968, leave=0.5, reach=0.5}
  [647] = {accel=80, decel=80, tmax=11.488, leave=0.5, reach=0.5}
  [648] = {accel=80, decel=80, tmax=12.518, leave=0.5, reach=0.5}
  [649] = {accel=80, decel=80, tmax=14.195, leave=0.5, reach=0.5}
  [650] = {accel=80, decel=80, tmax=16.276, leave=0.5, reach=0.5}
  [651] = {accel=80, decel=80, tmax=18.289, leave=0.5, reach=0.5}
  [652] = {accel=80, decel=80, tmax=20.091, leave=0.5, reach=0.5}
  [653] = {accel=80, decel=80, tmax=20.067, leave=0.5, reach=0.5}
  [654] = {accel=80, decel=80, tmax=18.818, leave=0.5, reach=0.5}
  [655] = {accel=80, decel=80, tmax=16.047, leave=0.5, reach=0.5}
  [656] = {accel=80, decel=80, tmax=13.333, leave=0.5, reach=0.5}
  [657] = {accel=80, decel=80, tmax=10.788, leave=0.5, reach=0.5}
  [658] = {accel=80, decel=80, tmax=9.076, leave=0.5, reach=0.5}
  [659] = {accel=80, decel=80, tmax=8.226, leave=0.5, reach=0.5}
  [660] = {accel=80, decel=80, tmax=7.861, leave=0.5, reach=0.5}
  [661] = {accel=80, decel=80, tmax=8.323, leave=0.5, reach=0.5}
  [662] = {accel=80, decel=80, tmax=9.575, leave=0.5, reach=0.5}
  [663] = {accel=80, decel=80, tmax=11.409, leave=0.5, reach=0.5}
  [664] = {accel=80, decel=80, tmax=13.342, leave=0.5, reach=0.5}
  [665] = {accel=80, decel=80, tmax=14.835, leave=0.5, reach=0.5}
  [666] = {accel=80, decel=80, tmax=16.324, leave=0.5, reach=0.5}
  [667] = {accel=80, decel=80, tmax=16.912, leave=0.5, reach=0.5}
  [668] = {accel=80, decel=80, tmax=16.912, leave=0.5, reach=0.5}
  [669] = {accel=80, decel=80, tmax=16.324, leave=0.5, reach=0.5}
  [670] = {accel=80, decel=80, tmax=14.835, leave=0.5, reach=0.5}
  [671] = {accel=80, decel=80, tmax=13.342, leave=0.5, reach=0.5}
  [672] = {accel=80, decel=80, tmax=11.409, leave=0.5, reach=0.5}
  [673] = {accel=80, decel=80, tmax=9.575, leave=0.5, reach=0.5}
  [674] = {accel=80, decel=80, tmax=8.323, leave=0.5, reach=0.5}
  [675] = {accel=80, decel=80, tmax=7.861, leave=0.5, reach=0.5}
  [676] = {accel=80, decel=80, tmax=8.226, leave=0.5, reach=0.5}
  [677] = {accel=80, decel=80, tmax=9.076, leave=0.5, reach=0.5}
  [678] = {accel=80, decel=80, tmax=10.788, leave=0.5, reach=0.5}
  [679] = {accel=80, decel=80, tmax=13.333, leave=0.5, reach=0.5}
  [680] = {accel=80, decel=80, tmax=16.047, leave=0.5, reach=0.5}
  [681] = {accel=80, decel=80, tmax=18.818, leave=0.5, reach=0.5}
  [682] = {accel=80, decel=80, tmax=20.067, leave=0.5, reach=0.5}
  [683] = {accel=80, decel=80, tmax=20.091, leave=0.5, reach=0.5}
  [684] = {accel=80, decel=80, tmax=18.289, leave=0.5, reach=0.5}
  [685] = {accel=80, decel=80, tmax=16.276, leave=0.5, reach=0.5}
  [686] = {accel=80, decel=80, tmax=14.195, leave=0.5, reach=0.5}
  [687] = {accel=80, decel=80, tmax=12.518, leave=0.5, reach=0.5}
  [688] = {accel=80, decel=80, tmax=11.488, leave=0.5, reach=0.5}
  [689] = {accel=80, decel=80, tmax=9.968, leave=0.5, reach=0.5}
  [690] = {accel=80, decel=80, tmax=8.512, leave=0.5, reach=0.5}
  [691] = {accel=80, decel=80, tmax=7.904, leave=0.5, reach=0.5}
  [692] = {accel=80, decel=80, tmax=9.015, leave=0.5, reach=0.5}
  [693] = {accel=80, decel=80, tmax=12.173, leave=0.5, reach=0.5}
  [694] = {accel=80, decel=80, tmax=16.689, leave=0.5, reach=0.5}
  [695] = {accel=80, decel=80, tmax=24.489, leave=0.5, reach=0.5}
  [696] = {accel=80, decel=80, tmax=27.687, leave=0.5, reach=0.5}
  [697] = {accel=80, decel=80, tmax=28.756, leave=0.5, reach=0.5}
  [698] = {accel=80, decel=80, tmax=25.104, leave=0.5, reach=0.5}
  [699] = {accel=80, decel=80, tmax=20.378, leave=0.5, reach=0.5}
  [700] = {accel=80, decel=80, tmax=16.152, leave=0.5, reach=0.5}
  [701] = {accel=80, decel=80, tmax=14.257, leave=0.5, reach=0.5}
  [702] = {accel=80, decel=80, tmax=14.258, leave=0.5, reach=0.5}
  [703] = {accel=80, decel=80, tmax=10.629, leave=0.5, reach=0.5}
  [704] = {accel=80, decel=80, tmax=7.443, leave=0.5, reach=0.5}
  [705] = {accel=80, decel=80, tmax=7.277, leave=0.5, reach=0.5}
  [706] = {accel=80, decel=80, tmax=9.932, leave=0.5, reach=0.5}
  [707] = {accel=80, decel=80, tmax=14.592, leave=0.5, reach=0.5}
  [708] = {accel=80, decel=80, tmax=12.487, leave=0.5, reach=0.5}
  [709] = {accel=80, decel=80, tmax=8.293, leave=0.5, reach=0.5}
  [710] = {accel=80, decel=80, tmax=8.474, leave=0.5, reach=0.5}
  [711] = {accel=80, decel=80, tmax=10.22, leave=0.5, reach=0.5}
  [712] = {accel=80, decel=80, tmax=12.308, leave=0.5, reach=0.5}
  [713] = {accel=80, decel=80, tmax=12.937, leave=0.5, reach=0.5}
  [714] = {accel=80, decel=80, tmax=13.257, leave=0.5, reach=0.5}
  [715] = {accel=80, decel=80, tmax=16.154, leave=0.5, reach=0.5}
  [716] = {accel=80, decel=80, tmax=18.767, leave=0.5, reach=0.5}
  [717] = {accel=80, decel=80, tmax=24.735, leave=0.5, reach=0.5}
  [718] = {accel=80, decel=80, tmax=25.595, leave=0.5, reach=0.5}
  [719] = {accel=80, decel=80, tmax=21.514, leave=0.5, reach=0.5}
  [720] = {accel=80, decel=80, tmax=17.816, leave=0.5, reach=0.5}
  [721] = {accel=80, decel=80, tmax=12.415, leave=0.5, reach=0.5}
  [722] = {accel=80, decel=80, tmax=9.135, leave=0.5, reach=0.5}
  [723] = {accel=80, decel=80, tmax=7.873, leave=0.5, reach=0.5}
  [724] = {accel=80, decel=80, tmax=8.361, leave=0.5, reach=0.5}
  [725] = {accel=80, decel=80, tmax=9.787, leave=0.5, reach=0.5}
  [726] = {accel=80, decel=80, tmax=11.5, leave=0.5, reach=0.5}
  [727] = {accel=80, decel=80, tmax=12.699, leave=0.5, reach=0.5}
  [728] = {accel=80, decel=80, tmax=13.935, leave=0.5, reach=0.5}
  [729] = {accel=80, decel=80, tmax=15.031, leave=0.5, reach=0.5}
  [730] = {accel=80, decel=80, tmax=16.479, leave=0.5, reach=0.5}
  [731] = {accel=80, decel=80, tmax=17.91, leave=0.5, reach=0.5}
  [732] = {accel=80, decel=80, tmax=18.011, leave=0.5, reach=0.5}
  [733] = {accel=80, decel=80, tmax=17.602, leave=0.5, reach=0.5}
  [734] = {accel=80, decel=80, tmax=15.847, leave=0.5, reach=0.5}
  [735] = {accel=80, decel=80, tmax=13.358, leave=0.5, reach=0.5}
  [736] = {accel=80, decel=80, tmax=11.095, leave=0.5, reach=0.5}
  [737] = {accel=80, decel=80, tmax=9.508, leave=0.5, reach=0.5}
  [738] = {accel=80, decel=80, tmax=8.34, leave=0.5, reach=0.5}
  [739] = {accel=80, decel=80, tmax=8.222, leave=0.5, reach=0.5}
  [740] = {accel=80, decel=80, tmax=8.676, leave=0.5, reach=0.5}
  [741] = {accel=80, decel=80, tmax=10.107, leave=0.5, reach=0.5}
  [742] = {accel=80, decel=80, tmax=12.173, leave=0.5, reach=0.5}
  [743] = {accel=80, decel=80, tmax=14.073, leave=0.5, reach=0.5}
  [744] = {accel=80, decel=80, tmax=15.651, leave=0.5, reach=0.5}
  [745] = {accel=80, decel=80, tmax=16.897, leave=0.5, reach=0.5}
  [746] = {accel=80, decel=80, tmax=18.883, leave=0.5, reach=0.5}
  [747] = {accel=80, decel=80, tmax=18.883, leave=0.5, reach=0.5}
  [748] = {accel=80, decel=80, tmax=16.897, leave=0.5, reach=0.5}
  [749] = {accel=80, decel=80, tmax=15.651, leave=0.5, reach=0.5}
  [750] = {accel=80, decel=80, tmax=14.073, leave=0.5, reach=0.5}
  [751] = {accel=80, decel=80, tmax=12.173, leave=0.5, reach=0.5}
  [752] = {accel=80, decel=80, tmax=10.107, leave=0.5, reach=0.5}
  [753] = {accel=80, decel=80, tmax=8.676, leave=0.5, reach=0.5}
  [754] = {accel=80, decel=80, tmax=8.222, leave=0.5, reach=0.5}
  [755] = {accel=80, decel=80, tmax=8.34, leave=0.5, reach=0.5}
  [756] = {accel=80, decel=80, tmax=9.508, leave=0.5, reach=0.5}
  [757] = {accel=80, decel=80, tmax=11.095, leave=0.5, reach=0.5}
  [758] = {accel=80, decel=80, tmax=13.358, leave=0.5, reach=0.5}
  [759] = {accel=80, decel=80, tmax=15.847, leave=0.5, reach=0.5}
  [760] = {accel=80, decel=80, tmax=17.602, leave=0.5, reach=0.5}
  [761] = {accel=80, decel=80, tmax=18.011, leave=0.5, reach=0.5}
  [762] = {accel=80, decel=80, tmax=17.91, leave=0.5, reach=0.5}
  [763] = {accel=80, decel=80, tmax=16.479, leave=0.5, reach=0.5}
  [764] = {accel=80, decel=80, tmax=15.031, leave=0.5, reach=0.5}
  [765] = {accel=80, decel=80, tmax=13.935, leave=0.5, reach=0.5}
  [766] = {accel=80, decel=80, tmax=12.699, leave=0.5, reach=0.5}
  [767] = {accel=80, decel=80, tmax=11.5, leave=0.5, reach=0.5}
  [768] = {accel=80, decel=80, tmax=9.787, leave=0.5, reach=0.5}
  [769] = {accel=80, decel=80, tmax=8.361, leave=0.5, reach=0.5}
  [770] = {accel=80, decel=80, tmax=7.873, leave=0.5, reach=0.5}
  [771] = {accel=80, decel=80, tmax=9.135, leave=0.5, reach=0.5}
  [772] = {accel=80, decel=80, tmax=12.415, leave=0.5, reach=0.5}
  [773] = {accel=80, decel=80, tmax=17.816, leave=0.5, reach=0.5}
  [774] = {accel=80, decel=80, tmax=21.514, leave=0.5, reach=0.5}
  [775] = {accel=80, decel=80, tmax=25.595, leave=0.5, reach=0.5}
  [776] = {accel=80, decel=80, tmax=24.735, leave=0.5, reach=0.5}
  [777] = {accel=80, decel=80, tmax=18.767, leave=0.5, reach=0.5}
  [778] = {accel=80, decel=80, tmax=16.154, leave=0.5, reach=0.5}
  [779] = {accel=80, decel=80, tmax=13.257, leave=0.5, reach=0.5}
  [780] = {accel=80, decel=80, tmax=12.937, leave=0.5, reach=0.5}
  [781] = {accel=80, decel=80, tmax=12.308, leave=0.5, reach=0.5}
  [782] = {accel=80, decel=80, tmax=10.22, leave=0.5, reach=0.5}
  [783] = {accel=80, decel=80, tmax=8.474, leave=0.5, reach=0.5}
  [784] = {accel=80, decel=80, tmax=8.293, leave=0.5, reach=0.5}
  [785] = {accel=80, decel=80, tmax=12.487, leave=0.5, reach=0.5}
  [786] = {accel=80, decel=80, tmax=10.71, leave=0.5, reach=0.5}
  [787] = {accel=80, decel=80, tmax=7.065, leave=0.5, reach=0.5}
  [788] = {accel=80, decel=80, tmax=6.813, leave=0.5, reach=0.5}
  [789] = {accel=80, decel=80, tmax=8.782, leave=0.5, reach=0.5}
  [790] = {accel=80, decel=80, tmax=12.532, leave=0.5, reach=0.5}
  [791] = {accel=80, decel=80, tmax=12.837, leave=0.5, reach=0.5}
  [792] = {accel=80, decel=80, tmax=12.393, leave=0.5, reach=0.5}
  [793] = {accel=80, decel=80, tmax=13.955, leave=0.5, reach=0.5}
  [794] = {accel=80, decel=80, tmax=15.754, leave=0.5, reach=0.5}
  [795] = {accel=80, decel=80, tmax=17.714, leave=0.5, reach=0.5}
  [796] = {accel=80, decel=80, tmax=20.079, leave=0.5, reach=0.5}
  [797] = {accel=80, decel=80, tmax=21.09, leave=0.5, reach=0.5}
  [798] = {accel=80, decel=80, tmax=20.54, leave=0.5, reach=0.5}
  [799] = {accel=80, decel=80, tmax=17.144, leave=0.5, reach=0.5}
  [800] = {accel=80, decel=80, tmax=13.335, leave=0.5, reach=0.5}
  [801] = {accel=80, decel=80, tmax=9.695, leave=0.5, reach=0.5}
  [802] = {accel=80, decel=80, tmax=7.477, leave=0.5, reach=0.5}
  [803] = {accel=80, decel=80, tmax=7.364, leave=0.5, reach=0.5}
  [804] = {accel=80, decel=80, tmax=8.691, leave=0.5, reach=0.5}
  [805] = {accel=80, decel=80, tmax=10.553, leave=0.5, reach=0.5}
  [806] = {accel=80, decel=80, tmax=11.822, leave=0.5, reach=0.5}
  [807] = {accel=80, decel=80, tmax=12.849, leave=0.5, reach=0.5}
  [808] = {accel=80, decel=80, tmax=14.388, leave=0.5, reach=0.5}
  [809] = {accel=80, decel=80, tmax=15.735, leave=0.5, reach=0.5}
  [810] = {accel=80, decel=80, tmax=17.331, leave=0.5, reach=0.5}
  [811] = {accel=80, decel=80, tmax=17.689, leave=0.5, reach=0.5}
  [812] = {accel=80, decel=80, tmax=17.183, leave=0.5, reach=0.5}
  [813] = {accel=80, decel=80, tmax=15.424, leave=0.5, reach=0.5}
  [814] = {accel=80, decel=80, tmax=13.165, leave=0.5, reach=0.5}
  [815] = {accel=80, decel=80, tmax=11.094, leave=0.5, reach=0.5}
  [816] = {accel=80, decel=80, tmax=9.231, leave=0.5, reach=0.5}
  [817] = {accel=80, decel=80, tmax=8.368, leave=0.5, reach=0.5}
  [818] = {accel=80, decel=80, tmax=8.075, leave=0.5, reach=0.5}
  [819] = {accel=80, decel=80, tmax=8.675, leave=0.5, reach=0.5}
  [820] = {accel=80, decel=80, tmax=9.924, leave=0.5, reach=0.5}
  [821] = {accel=80, decel=80, tmax=11.89, leave=0.5, reach=0.5}
  [822] = {accel=80, decel=80, tmax=14.316, leave=0.5, reach=0.5}
  [823] = {accel=80, decel=80, tmax=16.329, leave=0.5, reach=0.5}
  [824] = {accel=80, decel=80, tmax=17.996, leave=0.5, reach=0.5}
  [825] = {accel=80, decel=80, tmax=18.579, leave=0.5, reach=0.5}
  [826] = {accel=80, decel=80, tmax=18.579, leave=0.5, reach=0.5}
  [827] = {accel=80, decel=80, tmax=17.996, leave=0.5, reach=0.5}
  [828] = {accel=80, decel=80, tmax=16.329, leave=0.5, reach=0.5}
  [829] = {accel=80, decel=80, tmax=14.316, leave=0.5, reach=0.5}
  [830] = {accel=80, decel=80, tmax=11.89, leave=0.5, reach=0.5}
  [831] = {accel=80, decel=80, tmax=9.924, leave=0.5, reach=0.5}
  [832] = {accel=80, decel=80, tmax=8.675, leave=0.5, reach=0.5}
  [833] = {accel=80, decel=80, tmax=8.075, leave=0.5, reach=0.5}
  [834] = {accel=80, decel=80, tmax=8.368, leave=0.5, reach=0.5}
  [835] = {accel=80, decel=80, tmax=9.231, leave=0.5, reach=0.5}
  [836] = {accel=80, decel=80, tmax=11.094, leave=0.5, reach=0.5}
  [837] = {accel=80, decel=80, tmax=13.165, leave=0.5, reach=0.5}
  [838] = {accel=80, decel=80, tmax=15.424, leave=0.5, reach=0.5}
  [839] = {accel=80, decel=80, tmax=17.183, leave=0.5, reach=0.5}
  [840] = {accel=80, decel=80, tmax=17.689, leave=0.5, reach=0.5}
  [841] = {accel=80, decel=80, tmax=17.331, leave=0.5, reach=0.5}
  [842] = {accel=80, decel=80, tmax=15.735, leave=0.5, reach=0.5}
  [843] = {accel=80, decel=80, tmax=14.388, leave=0.5, reach=0.5}
  [844] = {accel=80, decel=80, tmax=12.849, leave=0.5, reach=0.5}
  [845] = {accel=80, decel=80, tmax=11.822, leave=0.5, reach=0.5}
  [846] = {accel=80, decel=80, tmax=10.553, leave=0.5, reach=0.5}
  [847] = {accel=80, decel=80, tmax=8.691, leave=0.5, reach=0.5}
  [848] = {accel=80, decel=80, tmax=7.364, leave=0.5, reach=0.5}
  [849] = {accel=80, decel=80, tmax=7.477, leave=0.5, reach=0.5}
  [850] = {accel=80, decel=80, tmax=9.695, leave=0.5, reach=0.5}
  [851] = {accel=80, decel=80, tmax=13.335, leave=0.5, reach=0.5}
  [852] = {accel=80, decel=80, tmax=17.144, leave=0.5, reach=0.5}
  [853] = {accel=80, decel=80, tmax=20.54, leave=0.5, reach=0.5}
  [854] = {accel=80, decel=80, tmax=21.09, leave=0.5, reach=0.5}
  [855] = {accel=80, decel=80, tmax=20.079, leave=0.5, reach=0.5}
  [856] = {accel=80, decel=80, tmax=17.714, leave=0.5, reach=0.5}
  [857] = {accel=80, decel=80, tmax=15.754, leave=0.5, reach=0.5}
  [858] = {accel=80, decel=80, tmax=13.955, leave=0.5, reach=0.5}
  [859] = {accel=80, decel=80, tmax=12.393, leave=0.5, reach=0.5}
  [860] = {accel=80, decel=80, tmax=12.837, leave=0.5, reach=0.5}
  [861] = {accel=80, decel=80, tmax=12.532, leave=0.5, reach=0.5}
  [862] = {accel=80, decel=80, tmax=8.782, leave=0.5, reach=0.5}
  [863] = {accel=80, decel=80, tmax=6.813, leave=0.5, reach=0.5}
  [864] = {accel=80, decel=80, tmax=7.065, leave=0.5, reach=0.5}
  [865] = {accel=80, decel=80, tmax=7.364, leave=0.5, reach=0.5}
  [866] = {accel=80, decel=80, tmax=6.776, leave=0.5, reach=0.5}
  [867] = {accel=80, decel=80, tmax=6.69, leave=0.5, reach=0.5}
  [868] = {accel=80, decel=80, tmax=9.392, leave=0.5, reach=0.5}
  [869] = {accel=80, decel=80, tmax=11.483, leave=0.5, reach=0.5}
  [870] = {accel=80, decel=80, tmax=9.789, leave=0.5, reach=0.5}
  [871] = {accel=80, decel=80, tmax=9.637, leave=0.5, reach=0.5}
  [872] = {accel=80, decel=80, tmax=10.361, leave=0.5, reach=0.5}
  [873] = {accel=80, decel=80, tmax=12.829, leave=0.5, reach=0.5}
  [874] = {accel=80, decel=80, tmax=15.481, leave=0.5, reach=0.5}
  [875] = {accel=80, decel=80, tmax=17.133, leave=0.5, reach=0.5}
  [876] = {accel=80, decel=80, tmax=18.371, leave=0.5, reach=0.5}
  [877] = {accel=80, decel=80, tmax=17.116, leave=0.5, reach=0.5}
  [878] = {accel=80, decel=80, tmax=15.677, leave=0.5, reach=0.5}
  [879] = {accel=80, decel=80, tmax=12.794, leave=0.5, reach=0.5}
  [880] = {accel=80, decel=80, tmax=9.787, leave=0.5, reach=0.5}
  [881] = {accel=80, decel=80, tmax=7.974, leave=0.5, reach=0.5}
  [882] = {accel=80, decel=80, tmax=7.593, leave=0.5, reach=0.5}
  [883] = {accel=80, decel=80, tmax=8.547, leave=0.5, reach=0.5}
  [884] = {accel=80, decel=80, tmax=10.746, leave=0.5, reach=0.5}
  [885] = {accel=80, decel=80, tmax=12.116, leave=0.5, reach=0.5}
  [886] = {accel=80, decel=80, tmax=12.313, leave=0.5, reach=0.5}
  [887] = {accel=80, decel=80, tmax=12.805, leave=0.5, reach=0.5}
  [888] = {accel=80, decel=80, tmax=13.735, leave=0.5, reach=0.5}
  [889] = {accel=80, decel=80, tmax=14.936, leave=0.5, reach=0.5}
  [890] = {accel=80, decel=80, tmax=15.27, leave=0.5, reach=0.5}
  [891] = {accel=80, decel=80, tmax=15.248, leave=0.5, reach=0.5}
  [892] = {accel=80, decel=80, tmax=14.588, leave=0.5, reach=0.5}
  [893] = {accel=80, decel=80, tmax=12.515, leave=0.5, reach=0.5}
  [894] = {accel=80, decel=80, tmax=11.03, leave=0.5, reach=0.5}
  [895] = {accel=80, decel=80, tmax=9.508, leave=0.5, reach=0.5}
  [896] = {accel=80, decel=80, tmax=8.591, leave=0.5, reach=0.5}
  [897] = {accel=80, decel=80, tmax=8.485, leave=0.5, reach=0.5}
  [898] = {accel=80, decel=80, tmax=8.788, leave=0.5, reach=0.5}
  [899] = {accel=80, decel=80, tmax=9.942, leave=0.5, reach=0.5}
  [900] = {accel=80, decel=80, tmax=11.626, leave=0.5, reach=0.5}
  [901] = {accel=80, decel=80, tmax=13.543, leave=0.5, reach=0.5}
  [902] = {accel=80, decel=80, tmax=15.037, leave=0.5, reach=0.5}
  [903] = {accel=80, decel=80, tmax=16.214, leave=0.5, reach=0.5}
  [904] = {accel=80, decel=80, tmax=17.06, leave=0.5, reach=0.5}
  [905] = {accel=80, decel=80, tmax=17.06, leave=0.5, reach=0.5}
  [906] = {accel=80, decel=80, tmax=16.214, leave=0.5, reach=0.5}
  [907] = {accel=80, decel=80, tmax=15.037, leave=0.5, reach=0.5}
  [908] = {accel=80, decel=80, tmax=13.543, leave=0.5, reach=0.5}
  [909] = {accel=80, decel=80, tmax=11.626, leave=0.5, reach=0.5}
  [910] = {accel=80, decel=80, tmax=9.942, leave=0.5, reach=0.5}
  [911] = {accel=80, decel=80, tmax=8.788, leave=0.5, reach=0.5}
  [912] = {accel=80, decel=80, tmax=8.485, leave=0.5, reach=0.5}
  [913] = {accel=80, decel=80, tmax=8.591, leave=0.5, reach=0.5}
  [914] = {accel=80, decel=80, tmax=9.508, leave=0.5, reach=0.5}
  [915] = {accel=80, decel=80, tmax=11.03, leave=0.5, reach=0.5}
  [916] = {accel=80, decel=80, tmax=12.515, leave=0.5, reach=0.5}
  [917] = {accel=80, decel=80, tmax=14.588, leave=0.5, reach=0.5}
  [918] = {accel=80, decel=80, tmax=15.248, leave=0.5, reach=0.5}
  [919] = {accel=80, decel=80, tmax=15.27, leave=0.5, reach=0.5}
  [920] = {accel=80, decel=80, tmax=14.936, leave=0.5, reach=0.5}
  [921] = {accel=80, decel=80, tmax=13.735, leave=0.5, reach=0.5}
  [922] = {accel=80, decel=80, tmax=12.805, leave=0.5, reach=0.5}
  [923] = {accel=80, decel=80, tmax=12.313, leave=0.5, reach=0.5}
  [924] = {accel=80, decel=80, tmax=12.116, leave=0.5, reach=0.5}
  [925] = {accel=80, decel=80, tmax=10.746, leave=0.5, reach=0.5}
  [926] = {accel=80, decel=80, tmax=8.547, leave=0.5, reach=0.5}
  [927] = {accel=80, decel=80, tmax=7.593, leave=0.5, reach=0.5}
  [928] = {accel=80, decel=80, tmax=7.974, leave=0.5, reach=0.5}
  [929] = {accel=80, decel=80, tmax=9.787, leave=0.5, reach=0.5}
  [930] = {accel=80, decel=80, tmax=12.794, leave=0.5, reach=0.5}
  [931] = {accel=80, decel=80, tmax=15.677, leave=0.5, reach=0.5}
  [932] = {accel=80, decel=80, tmax=17.116, leave=0.5, reach=0.5}
  [933] = {accel=80, decel=80, tmax=18.371, leave=0.5, reach=0.5}
  [934] = {accel=80, decel=80, tmax=17.133, leave=0.5, reach=0.5}
  [935] = {accel=80, decel=80, tmax=15.481, leave=0.5, reach=0.5}
  [936] = {accel=80, decel=80, tmax=12.829, leave=0.5, reach=0.5}
  [937] = {accel=80, decel=80, tmax=10.361, leave=0.5, reach=0.5}
  [938] = {accel=80, decel=80, tmax=9.637, leave=0.5, reach=0.5}
  [939] = {accel=80, decel=80, tmax=9.789, leave=0.5, reach=0.5}
  [940] = {accel=80, decel=80, tmax=11.483, leave=0.5, reach=0.5}
  [941] = {accel=80, decel=80, tmax=9.392, leave=0.5, reach=0.5}
  [942] = {accel=80, decel=80, tmax=6.69, leave=0.5, reach=0.5}
  [943] = {accel=80, decel=80, tmax=6.776, leave=0.5, reach=0.5}
  [944] = {accel=80, decel=80, tmax=4.92, leave=0.5, reach=0.5}
  [945] = {accel=80, decel=80, tmax=4.399, leave=0.5, reach=0.5}
  [946] = {accel=80, decel=80, tmax=6.338, leave=0.5, reach=0.5}
  [947] = {accel=80, decel=80, tmax=10.204, leave=0.5, reach=0.5}
  [948] = {accel=80, decel=80, tmax=12.733, leave=0.5, reach=0.5}
  [949] = {accel=80, decel=80, tmax=10.189, leave=0.5, reach=0.5}
  [950] = {accel=80, decel=80, tmax=9.004, leave=0.5, reach=0.5}
  [951] = {accel=80, decel=80, tmax=9.559, leave=0.5, reach=0.5}
  [952] = {accel=80, decel=80, tmax=11.37, leave=0.5, reach=0.5}
  [953] = {accel=80, decel=80, tmax=12.953, leave=0.5, reach=0.5}
  [954] = {accel=80, decel=80, tmax=13.825, leave=0.5, reach=0.5}
  [955] = {accel=80, decel=80, tmax=15.163, leave=0.5, reach=0.5}
  [956] = {accel=80, decel=80, tmax=15.256, leave=0.5, reach=0.5}
  [957] = {accel=80, decel=80, tmax=14.425, leave=0.5, reach=0.5}
  [958] = {accel=80, decel=80, tmax=12.345, leave=0.5, reach=0.5}
  [959] = {accel=80, decel=80, tmax=10.02, leave=0.5, reach=0.5}
  [960] = {accel=80, decel=80, tmax=7.802, leave=0.5, reach=0.5}
  [961] = {accel=80, decel=80, tmax=6.952, leave=0.5, reach=0.5}
  [962] = {accel=80, decel=80, tmax=7.453, leave=0.5, reach=0.5}
  [963] = {accel=80, decel=80, tmax=9.277, leave=0.5, reach=0.5}
  [964] = {accel=80, decel=80, tmax=11.196, leave=0.5, reach=0.5}
  [965] = {accel=80, decel=80, tmax=11.817, leave=0.5, reach=0.5}
  [966] = {accel=80, decel=80, tmax=11.985, leave=0.5, reach=0.5}
  [967] = {accel=80, decel=80, tmax=12.678, leave=0.5, reach=0.5}
  [968] = {accel=80, decel=80, tmax=13.77, leave=0.5, reach=0.5}
  [969] = {accel=80, decel=80, tmax=14.249, leave=0.5, reach=0.5}
  [970] = {accel=80, decel=80, tmax=14.561, leave=0.5, reach=0.5}
  [971] = {accel=80, decel=80, tmax=13.657, leave=0.5, reach=0.5}
  [972] = {accel=80, decel=80, tmax=12.216, leave=0.5, reach=0.5}
  [973] = {accel=80, decel=80, tmax=10.553, leave=0.5, reach=0.5}
  [974] = {accel=80, decel=80, tmax=9.156, leave=0.5, reach=0.5}
  [975] = {accel=80, decel=80, tmax=8.496, leave=0.5, reach=0.5}
  [976] = {accel=80, decel=80, tmax=8.028, leave=0.5, reach=0.5}
  [977] = {accel=80, decel=80, tmax=8.46, leave=0.5, reach=0.5}
  [978] = {accel=80, decel=80, tmax=9.468, leave=0.5, reach=0.5}
  [979] = {accel=80, decel=80, tmax=11.19, leave=0.5, reach=0.5}
  [980] = {accel=80, decel=80, tmax=13.721, leave=0.5, reach=0.5}
  [981] = {accel=80, decel=80, tmax=15.814, leave=0.5, reach=0.5}
  [982] = {accel=80, decel=80, tmax=16.89, leave=0.5, reach=0.5}
  [983] = {accel=80, decel=80, tmax=17.466, leave=0.5, reach=0.5}
  [984] = {accel=80, decel=80, tmax=17.466, leave=0.5, reach=0.5}
  [985] = {accel=80, decel=80, tmax=16.89, leave=0.5, reach=0.5}
  [986] = {accel=80, decel=80, tmax=15.814, leave=0.5, reach=0.5}
  [987] = {accel=80, decel=80, tmax=13.721, leave=0.5, reach=0.5}
  [988] = {accel=80, decel=80, tmax=11.19, leave=0.5, reach=0.5}
  [989] = {accel=80, decel=80, tmax=9.468, leave=0.5, reach=0.5}
  [990] = {accel=80, decel=80, tmax=8.46, leave=0.5, reach=0.5}
  [991] = {accel=80, decel=80, tmax=8.028, leave=0.5, reach=0.5}
  [992] = {accel=80, decel=80, tmax=8.496, leave=0.5, reach=0.5}
  [993] = {accel=80, decel=80, tmax=9.156, leave=0.5, reach=0.5}
  [994] = {accel=80, decel=80, tmax=10.553, leave=0.5, reach=0.5}
  [995] = {accel=80, decel=80, tmax=12.216, leave=0.5, reach=0.5}
  [996] = {accel=80, decel=80, tmax=13.657, leave=0.5, reach=0.5}
  [997] = {accel=80, decel=80, tmax=14.561, leave=0.5, reach=0.5}
  [998] = {accel=80, decel=80, tmax=14.249, leave=0.5, reach=0.5}
  [999] = {accel=80, decel=80, tmax=13.77, leave=0.5, reach=0.5}
num K = 35
num nCountCycle = 1
public num nCurrentTraj = 1
num nCurtRadius
num nDistToOrign = 225.000310635
num nFileId
num nFileId2 = 1
num nHundredRead
num nHundredWrite
public num nMoveID = 4499
public num nPrdRadius = 50.0559565
num nPtBuffer = 500
num nPtOfTraj[16] = 4499
num nReadJnt = 2
public num nReadPtr = 499
public num nSpdOfTCP
public num nTabSpdCode
public num nThousandRead = 4
public num nThousandWrite = 4
num nTime[2]
  [0] = 1611.967
  [1] = -4198.782
public num nTotalTrajs = 1
public num nTrajofRead
num nWriteJnt = 2
public num nWritePtr = 499
public num nZshift = -50
pointRx pGrinding = {x=-120.922, y=100.599, z=77.126, rx=10.14, ry=-162.354, rz=-27, fatherId=fPrdFrame[0]}
pointRx pPBuff = {x=1609.294798, y=46.814741, z=58.995545, rx=0.56357, ry=179.576697, rz=17.423888, shoulder=lefty, elbow=epositive, wrist=wpositive, fatherId=world[0]}
pointRx pPointRead[1000]
  [0] = {x=-59.216, y=83.465, z=9.504, rx=-171.87, ry=-7.549, rz=153, fatherId=fPrdFrame[0]}
  [1] = {x=-62.022, y=83.462, z=9.914, rx=-171.863, ry=-7.996, rz=153, fatherId=fPrdFrame[0]}
  [2] = {x=-64.829, y=83.458, z=10.347, rx=-171.856, ry=-8.443, rz=153, fatherId=fPrdFrame[0]}
  [3] = {x=-67.636, y=83.455, z=10.804, rx=-171.848, ry=-8.891, rz=153, fatherId=fPrdFrame[0]}
  [4] = {x=-70.443, y=83.452, z=11.286, rx=-171.84, ry=-9.34, rz=153, fatherId=fPrdFrame[0]}
  [5] = {x=-73.25, y=83.448, z=11.791, rx=-171.831, ry=-9.789, rz=153, fatherId=fPrdFrame[0]}
  [6] = {x=-76.057, y=83.444, z=12.321, rx=-171.822, ry=-10.238, rz=153, fatherId=fPrdFrame[0]}
  [7] = {x=-78.863, y=83.44, z=12.875, rx=-171.813, ry=-10.688, rz=153, fatherId=fPrdFrame[0]}
  [8] = {x=-81.67, y=83.435, z=13.453, rx=-171.803, ry=-11.139, rz=153, fatherId=fPrdFrame[0]}
  [9] = {x=-84.477, y=83.431, z=14.056, rx=-171.792, ry=-11.591, rz=153, fatherId=fPrdFrame[0]}
  [10] = {x=-87.284, y=83.426, z=14.684, rx=-171.781, ry=-12.043, rz=153, fatherId=fPrdFrame[0]}
  [11] = {x=-90.091, y=83.421, z=15.336, rx=-171.77, ry=-12.496, rz=153, fatherId=fPrdFrame[0]}
  [12] = {x=-92.897, y=83.416, z=16.014, rx=-171.758, ry=-12.95, rz=153, fatherId=fPrdFrame[0]}
  [13] = {x=-95.704, y=83.411, z=16.716, rx=-171.746, ry=-13.405, rz=153, fatherId=fPrdFrame[0]}
  [14] = {x=-98.511, y=83.405, z=17.444, rx=-171.733, ry=-13.86, rz=153, fatherId=fPrdFrame[0]}
  [15] = {x=-101.318, y=83.4, z=18.197, rx=-171.72, ry=-14.317, rz=153, fatherId=fPrdFrame[0]}
  [16] = {x=-104.125, y=83.394, z=18.975, rx=-171.706, ry=-14.774, rz=153, fatherId=fPrdFrame[0]}
  [17] = {x=-106.932, y=83.388, z=19.779, rx=-171.692, ry=-15.232, rz=153, fatherId=fPrdFrame[0]}
  [18] = {x=-109.739, y=83.381, z=20.609, rx=-171.677, ry=-15.691, rz=153, fatherId=fPrdFrame[0]}
  [19] = {x=-112.545, y=83.375, z=21.465, rx=-171.662, ry=-16.152, rz=153, fatherId=fPrdFrame[0]}
  [20] = {x=-115.352, y=83.368, z=22.346, rx=-171.646, ry=-16.613, rz=153, fatherId=fPrdFrame[0]}
  [21] = {x=-118.159, y=83.361, z=23.255, rx=-171.629, ry=-17.076, rz=153, fatherId=fPrdFrame[0]}
  [22] = {x=-120.966, y=83.353, z=24.19, rx=-171.612, ry=-17.539, rz=153, fatherId=fPrdFrame[0]}
  [23] = {x=-120.959, y=86.228, z=24.64, rx=-171.321, ry=-17.555, rz=153, fatherId=fPrdFrame[0]}
  [24] = {x=-118.153, y=86.235, z=23.704, rx=-171.339, ry=-17.091, rz=153, fatherId=fPrdFrame[0]}
  [25] = {x=-115.346, y=86.242, z=22.795, rx=-171.356, ry=-16.628, rz=153, fatherId=fPrdFrame[0]}
  [26] = {x=-112.539, y=86.25, z=21.912, rx=-171.372, ry=-16.167, rz=153, fatherId=fPrdFrame[0]}
  [27] = {x=-109.732, y=86.256, z=21.055, rx=-171.388, ry=-15.706, rz=153, fatherId=fPrdFrame[0]}
  [28] = {x=-106.926, y=86.263, z=20.225, rx=-171.403, ry=-15.246, rz=153, fatherId=fPrdFrame[0]}
  [29] = {x=-104.119, y=86.269, z=19.42, rx=-171.418, ry=-14.788, rz=153, fatherId=fPrdFrame[0]}
  [30] = {x=-101.312, y=86.275, z=18.641, rx=-171.432, ry=-14.33, rz=153, fatherId=fPrdFrame[0]}
  [31] = {x=-98.506, y=86.281, z=17.887, rx=-171.446, ry=-13.873, rz=153, fatherId=fPrdFrame[0]}
  [32] = {x=-95.699, y=86.287, z=17.159, rx=-171.459, ry=-13.417, rz=153, fatherId=fPrdFrame[0]}
  [33] = {x=-92.892, y=86.293, z=16.456, rx=-171.472, ry=-12.962, rz=153, fatherId=fPrdFrame[0]}
  [34] = {x=-90.086, y=86.298, z=15.778, rx=-171.484, ry=-12.508, rz=153, fatherId=fPrdFrame[0]}
  [35] = {x=-87.279, y=86.303, z=15.125, rx=-171.496, ry=-12.054, rz=153, fatherId=fPrdFrame[0]}
  [36] = {x=-84.472, y=86.308, z=14.497, rx=-171.507, ry=-11.601, rz=153, fatherId=fPrdFrame[0]}
  [37] = {x=-81.666, y=86.312, z=13.893, rx=-171.518, ry=-11.149, rz=153, fatherId=fPrdFrame[0]}
  [38] = {x=-78.859, y=86.317, z=13.314, rx=-171.528, ry=-10.698, rz=153, fatherId=fPrdFrame[0]}
  [39] = {x=-76.052, y=86.321, z=12.759, rx=-171.538, ry=-10.247, rz=153, fatherId=fPrdFrame[0]}
  [40] = {x=-73.246, y=86.325, z=12.229, rx=-171.548, ry=-9.797, rz=153, fatherId=fPrdFrame[0]}
  [41] = {x=-70.439, y=86.329, z=11.723, rx=-171.556, ry=-9.348, rz=153, fatherId=fPrdFrame[0]}
  [42] = {x=-67.633, y=86.333, z=11.242, rx=-171.565, ry=-8.899, rz=153, fatherId=fPrdFrame[0]}
  [43] = {x=-64.826, y=86.336, z=10.784, rx=-171.573, ry=-8.451, rz=153, fatherId=fPrdFrame[0]}
  [44] = {x=-62.019, y=86.34, z=10.35, rx=-171.581, ry=-8.003, rz=153, fatherId=fPrdFrame[0]}
  [45] = {x=-59.213, y=86.343, z=9.94, rx=-171.588, ry=-7.556, rz=153, fatherId=fPrdFrame[0]}
  [46] = {x=-56.406, y=86.346, z=9.554, rx=-171.595, ry=-7.109, rz=153, fatherId=fPrdFrame[0]}
  [47] = {x=-53.599, y=86.348, z=9.192, rx=-171.601, ry=-6.663, rz=153, fatherId=fPrdFrame[0]}
  [48] = {x=-50.793, y=86.351, z=8.853, rx=-171.607, ry=-6.217, rz=153, fatherId=fPrdFrame[0]}
  [49] = {x=-47.986, y=86.353, z=8.538, rx=-171.612, ry=-5.771, rz=153, fatherId=fPrdFrame[0]}
  [50] = {x=-45.179, y=86.355, z=8.247, rx=-171.618, ry=-5.326, rz=153, fatherId=fPrdFrame[0]}
  [51] = {x=-42.373, y=86.358, z=7.979, rx=-171.622, ry=-4.881, rz=153, fatherId=fPrdFrame[0]}
  [52] = {x=-39.566, y=86.359, z=7.734, rx=-171.626, ry=-4.436, rz=153, fatherId=fPrdFrame[0]}
  [53] = {x=-36.76, y=86.361, z=7.513, rx=-171.63, ry=-3.992, rz=153, fatherId=fPrdFrame[0]}
  [54] = {x=-33.953, y=86.362, z=7.316, rx=-171.634, ry=-3.548, rz=153, fatherId=fPrdFrame[0]}
  [55] = {x=-31.146, y=86.364, z=7.141, rx=-171.637, ry=-3.104, rz=153, fatherId=fPrdFrame[0]}
  [56] = {x=-28.34, y=86.365, z=6.99, rx=-171.639, ry=-2.66, rz=153, fatherId=fPrdFrame[0]}
  [57] = {x=-25.533, y=86.366, z=6.863, rx=-171.642, ry=-2.217, rz=153, fatherId=fPrdFrame[0]}
  [58] = {x=-22.726, y=86.367, z=6.758, rx=-171.643, ry=-1.773, rz=153, fatherId=fPrdFrame[0]}
  [59] = {x=-19.92, y=86.367, z=6.677, rx=-171.645, ry=-1.33, rz=153, fatherId=fPrdFrame[0]}
  [60] = {x=-17.113, y=86.368, z=6.619, rx=-171.646, ry=-0.886, rz=153, fatherId=fPrdFrame[0]}
  [61] = {x=-14.307, y=86.368, z=6.584, rx=-171.646, ry=-0.443, rz=153, fatherId=fPrdFrame[0]}
  [62] = {x=-11.5, y=86.368, z=6.572, rx=-171.647, rz=153, fatherId=fPrdFrame[0]}
  [63] = {x=-8.693, y=86.368, z=6.584, rx=-171.646, ry=0.443, rz=153, fatherId=fPrdFrame[0]}
  [64] = {x=-5.887, y=86.368, z=6.619, rx=-171.646, ry=0.886, rz=153, fatherId=fPrdFrame[0]}
  [65] = {x=-3.08, y=86.367, z=6.677, rx=-171.645, ry=1.33, rz=153, fatherId=fPrdFrame[0]}
  [66] = {x=-0.274, y=86.367, z=6.758, rx=-171.643, ry=1.773, rz=153, fatherId=fPrdFrame[0]}
  [67] = {x=2.533, y=86.366, z=6.863, rx=-171.642, ry=2.217, rz=153, fatherId=fPrdFrame[0]}
  [68] = {x=5.34, y=86.365, z=6.99, rx=-171.639, ry=2.66, rz=153, fatherId=fPrdFrame[0]}
  [69] = {x=8.146, y=86.364, z=7.141, rx=-171.637, ry=3.104, rz=153, fatherId=fPrdFrame[0]}
  [70] = {x=10.953, y=86.362, z=7.316, rx=-171.634, ry=3.548, rz=153, fatherId=fPrdFrame[0]}
  [71] = {x=13.76, y=86.361, z=7.513, rx=-171.63, ry=3.992, rz=153, fatherId=fPrdFrame[0]}
  [72] = {x=16.566, y=86.359, z=7.734, rx=-171.626, ry=4.436, rz=153, fatherId=fPrdFrame[0]}
  [73] = {x=19.373, y=86.358, z=7.979, rx=-171.622, ry=4.881, rz=153, fatherId=fPrdFrame[0]}
  [74] = {x=22.179, y=86.355, z=8.247, rx=-171.618, ry=5.326, rz=153, fatherId=fPrdFrame[0]}
  [75] = {x=24.986, y=86.353, z=8.538, rx=-171.612, ry=5.771, rz=153, fatherId=fPrdFrame[0]}
  [76] = {x=27.793, y=86.351, z=8.853, rx=-171.607, ry=6.217, rz=153, fatherId=fPrdFrame[0]}
  [77] = {x=30.599, y=86.348, z=9.192, rx=-171.601, ry=6.663, rz=153, fatherId=fPrdFrame[0]}
  [78] = {x=33.406, y=86.346, z=9.554, rx=-171.595, ry=7.109, rz=153, fatherId=fPrdFrame[0]}
  [79] = {x=36.213, y=86.343, z=9.94, rx=-171.588, ry=7.556, rz=153, fatherId=fPrdFrame[0]}
  [80] = {x=39.019, y=86.34, z=10.35, rx=-171.581, ry=8.003, rz=153, fatherId=fPrdFrame[0]}
  [81] = {x=41.826, y=86.336, z=10.784, rx=-171.573, ry=8.451, rz=153, fatherId=fPrdFrame[0]}
  [82] = {x=44.633, y=86.333, z=11.242, rx=-171.565, ry=8.899, rz=153, fatherId=fPrdFrame[0]}
  [83] = {x=47.439, y=86.329, z=11.723, rx=-171.556, ry=9.348, rz=153, fatherId=fPrdFrame[0]}
  [84] = {x=50.246, y=86.325, z=12.229, rx=-171.548, ry=9.797, rz=153, fatherId=fPrdFrame[0]}
  [85] = {x=53.052, y=86.321, z=12.759, rx=-171.538, ry=10.247, rz=153, fatherId=fPrdFrame[0]}
  [86] = {x=55.859, y=86.317, z=13.314, rx=-171.528, ry=10.698, rz=153, fatherId=fPrdFrame[0]}
  [87] = {x=58.666, y=86.312, z=13.893, rx=-171.518, ry=11.149, rz=153, fatherId=fPrdFrame[0]}
  [88] = {x=61.472, y=86.308, z=14.497, rx=-171.507, ry=11.601, rz=153, fatherId=fPrdFrame[0]}
  [89] = {x=64.279, y=86.303, z=15.125, rx=-171.496, ry=12.054, rz=153, fatherId=fPrdFrame[0]}
  [90] = {x=67.086, y=86.298, z=15.778, rx=-171.484, ry=12.508, rz=153, fatherId=fPrdFrame[0]}
  [91] = {x=69.892, y=86.293, z=16.456, rx=-171.472, ry=12.962, rz=153, fatherId=fPrdFrame[0]}
  [92] = {x=72.699, y=86.287, z=17.159, rx=-171.459, ry=13.417, rz=153, fatherId=fPrdFrame[0]}
  [93] = {x=75.506, y=86.281, z=17.887, rx=-171.446, ry=13.873, rz=153, fatherId=fPrdFrame[0]}
  [94] = {x=78.312, y=86.275, z=18.641, rx=-171.432, ry=14.33, rz=153, fatherId=fPrdFrame[0]}
  [95] = {x=81.119, y=86.269, z=19.42, rx=-171.418, ry=14.788, rz=153, fatherId=fPrdFrame[0]}
  [96] = {x=83.926, y=86.263, z=20.225, rx=-171.403, ry=15.246, rz=153, fatherId=fPrdFrame[0]}
  [97] = {x=86.732, y=86.256, z=21.055, rx=-171.388, ry=15.706, rz=153, fatherId=fPrdFrame[0]}
  [98] = {x=89.539, y=86.25, z=21.912, rx=-171.372, ry=16.167, rz=153, fatherId=fPrdFrame[0]}
  [99] = {x=92.346, y=86.242, z=22.795, rx=-171.356, ry=16.628, rz=153, fatherId=fPrdFrame[0]}
  [100] = {x=95.153, y=86.235, z=23.704, rx=-171.339, ry=17.091, rz=153, fatherId=fPrdFrame[0]}
  [101] = {x=97.959, y=86.228, z=24.64, rx=-171.321, ry=17.555, rz=153, fatherId=fPrdFrame[0]}
  [102] = {x=97.952, y=89.102, z=25.105, rx=-171.029, ry=17.572, rz=153, fatherId=fPrdFrame[0]}
  [103] = {x=95.146, y=89.11, z=24.169, rx=-171.047, ry=17.108, rz=153, fatherId=fPrdFrame[0]}
  [104] = {x=92.339, y=89.117, z=23.259, rx=-171.065, ry=16.644, rz=153, fatherId=fPrdFrame[0]}
  [105] = {x=89.533, y=89.124, z=22.375, rx=-171.082, ry=16.182, rz=153, fatherId=fPrdFrame[0]}
  [106] = {x=86.726, y=89.132, z=21.517, rx=-171.098, ry=15.721, rz=153, fatherId=fPrdFrame[0]}
  [107] = {x=83.92, y=89.138, z=20.686, rx=-171.114, ry=15.261, rz=153, fatherId=fPrdFrame[0]}
  [108] = {x=81.113, y=89.145, z=19.88, rx=-171.129, ry=14.802, rz=153, fatherId=fPrdFrame[0]}
  [109] = {x=78.307, y=89.151, z=19.101, rx=-171.144, ry=14.343, rz=153, fatherId=fPrdFrame[0]}
  [110] = {x=75.5, y=89.157, z=18.346, rx=-171.158, ry=13.886, rz=153, fatherId=fPrdFrame[0]}
  [111] = {x=72.694, y=89.163, z=17.617, rx=-171.172, ry=13.43, rz=153, fatherId=fPrdFrame[0]}
  [112] = {x=69.887, y=89.169, z=16.913, rx=-171.185, ry=12.974, rz=153, fatherId=fPrdFrame[0]}
  [113] = {x=67.081, y=89.174, z=16.235, rx=-171.198, ry=12.52, rz=153, fatherId=fPrdFrame[0]}
  [114] = {x=64.274, y=89.18, z=15.581, rx=-171.21, ry=12.066, rz=153, fatherId=fPrdFrame[0]}
  [115] = {x=61.468, y=89.185, z=14.952, rx=-171.222, ry=11.612, rz=153, fatherId=fPrdFrame[0]}
  [116] = {x=58.661, y=89.19, z=14.348, rx=-171.233, ry=11.16, rz=153, fatherId=fPrdFrame[0]}
  [117] = {x=55.855, y=89.194, z=13.768, rx=-171.244, ry=10.708, rz=153, fatherId=fPrdFrame[0]}
  [118] = {x=53.048, y=89.199, z=13.213, rx=-171.254, ry=10.257, rz=153, fatherId=fPrdFrame[0]}
  [119] = {x=50.242, y=89.203, z=12.683, rx=-171.264, ry=9.807, rz=153, fatherId=fPrdFrame[0]}
  [120] = {x=47.435, y=89.207, z=12.176, rx=-171.273, ry=9.357, rz=153, fatherId=fPrdFrame[0]}
  [121] = {x=44.629, y=89.211, z=11.694, rx=-171.282, ry=8.908, rz=153, fatherId=fPrdFrame[0]}
  [122] = {x=41.822, y=89.214, z=11.236, rx=-171.29, ry=8.459, rz=153, fatherId=fPrdFrame[0]}
  [123] = {x=39.016, y=89.218, z=10.802, rx=-171.298, ry=8.011, rz=153, fatherId=fPrdFrame[0]}
  [124] = {x=36.21, y=89.221, z=10.391, rx=-171.305, ry=7.563, rz=153, fatherId=fPrdFrame[0]}
  [125] = {x=33.403, y=89.224, z=10.005, rx=-171.312, ry=7.116, rz=153, fatherId=fPrdFrame[0]}
  [126] = {x=30.597, y=89.227, z=9.642, rx=-171.319, ry=6.669, rz=153, fatherId=fPrdFrame[0]}
  [127] = {x=27.79, y=89.229, z=9.303, rx=-171.325, ry=6.223, rz=153, fatherId=fPrdFrame[0]}
  [128] = {x=24.984, y=89.232, z=8.988, rx=-171.331, ry=5.777, rz=153, fatherId=fPrdFrame[0]}
  [129] = {x=22.177, y=89.234, z=8.696, rx=-171.336, ry=5.331, rz=153, fatherId=fPrdFrame[0]}
  [130] = {x=19.371, y=89.236, z=8.428, rx=-171.341, ry=4.886, rz=153, fatherId=fPrdFrame[0]}
  [131] = {x=16.564, y=89.238, z=8.184, rx=-171.345, ry=4.441, rz=153, fatherId=fPrdFrame[0]}
  [132] = {x=13.758, y=89.24, z=7.962, rx=-171.349, ry=3.996, rz=153, fatherId=fPrdFrame[0]}
  [133] = {x=10.952, y=89.241, z=7.764, rx=-171.353, ry=3.551, rz=153, fatherId=fPrdFrame[0]}
  [134] = {x=8.145, y=89.243, z=7.59, rx=-171.356, ry=3.107, rz=153, fatherId=fPrdFrame[0]}
  [135] = {x=5.339, y=89.244, z=7.439, rx=-171.359, ry=2.663, rz=153, fatherId=fPrdFrame[0]}
  [136] = {x=2.532, y=89.245, z=7.311, rx=-171.361, ry=2.219, rz=153, fatherId=fPrdFrame[0]}
  [137] = {x=-0.274, y=89.246, z=7.206, rx=-171.363, ry=1.775, rz=153, fatherId=fPrdFrame[0]}
  [138] = {x=-3.081, y=89.246, z=7.125, rx=-171.364, ry=1.331, rz=153, fatherId=fPrdFrame[0]}
  [139] = {x=-5.887, y=89.247, z=7.067, rx=-171.365, ry=0.887, rz=153, fatherId=fPrdFrame[0]}
  [140] = {x=-8.694, y=89.247, z=7.032, rx=-171.366, ry=0.444, rz=153, fatherId=fPrdFrame[0]}
  [141] = {x=-11.5, y=89.247, z=7.02, rx=-171.366, rz=153, fatherId=fPrdFrame[0]}
  [142] = {x=-14.306, y=89.247, z=7.032, rx=-171.366, ry=-0.444, rz=153, fatherId=fPrdFrame[0]}
  [143] = {x=-17.113, y=89.247, z=7.067, rx=-171.365, ry=-0.887, rz=153, fatherId=fPrdFrame[0]}
  [144] = {x=-19.919, y=89.246, z=7.125, rx=-171.364, ry=-1.331, rz=153, fatherId=fPrdFrame[0]}
  [145] = {x=-22.726, y=89.246, z=7.206, rx=-171.363, ry=-1.775, rz=153, fatherId=fPrdFrame[0]}
  [146] = {x=-25.532, y=89.245, z=7.311, rx=-171.361, ry=-2.219, rz=153, fatherId=fPrdFrame[0]}
  [147] = {x=-28.339, y=89.244, z=7.439, rx=-171.359, ry=-2.663, rz=153, fatherId=fPrdFrame[0]}
  [148] = {x=-31.145, y=89.243, z=7.59, rx=-171.356, ry=-3.107, rz=153, fatherId=fPrdFrame[0]}
  [149] = {x=-33.952, y=89.241, z=7.764, rx=-171.353, ry=-3.551, rz=153, fatherId=fPrdFrame[0]}
  [150] = {x=-36.758, y=89.24, z=7.962, rx=-171.349, ry=-3.996, rz=153, fatherId=fPrdFrame[0]}
  [151] = {x=-39.564, y=89.238, z=8.184, rx=-171.345, ry=-4.441, rz=153, fatherId=fPrdFrame[0]}
  [152] = {x=-42.371, y=89.236, z=8.428, rx=-171.341, ry=-4.886, rz=153, fatherId=fPrdFrame[0]}
  [153] = {x=-45.177, y=89.234, z=8.696, rx=-171.336, ry=-5.331, rz=153, fatherId=fPrdFrame[0]}
  [154] = {x=-47.984, y=89.232, z=8.988, rx=-171.331, ry=-5.777, rz=153, fatherId=fPrdFrame[0]}
  [155] = {x=-50.79, y=89.229, z=9.303, rx=-171.325, ry=-6.223, rz=153, fatherId=fPrdFrame[0]}
  [156] = {x=-53.597, y=89.227, z=9.642, rx=-171.319, ry=-6.669, rz=153, fatherId=fPrdFrame[0]}
  [157] = {x=-56.403, y=89.224, z=10.005, rx=-171.312, ry=-7.116, rz=153, fatherId=fPrdFrame[0]}
  [158] = {x=-59.21, y=89.221, z=10.391, rx=-171.305, ry=-7.563, rz=153, fatherId=fPrdFrame[0]}
  [159] = {x=-62.016, y=89.218, z=10.802, rx=-171.298, ry=-8.011, rz=153, fatherId=fPrdFrame[0]}
  [160] = {x=-64.822, y=89.214, z=11.236, rx=-171.29, ry=-8.459, rz=153, fatherId=fPrdFrame[0]}
  [161] = {x=-67.629, y=89.211, z=11.694, rx=-171.282, ry=-8.908, rz=153, fatherId=fPrdFrame[0]}
  [162] = {x=-70.435, y=89.207, z=12.176, rx=-171.273, ry=-9.357, rz=153, fatherId=fPrdFrame[0]}
  [163] = {x=-73.242, y=89.203, z=12.683, rx=-171.264, ry=-9.807, rz=153, fatherId=fPrdFrame[0]}
  [164] = {x=-76.048, y=89.199, z=13.213, rx=-171.254, ry=-10.257, rz=153, fatherId=fPrdFrame[0]}
  [165] = {x=-78.855, y=89.194, z=13.768, rx=-171.244, ry=-10.708, rz=153, fatherId=fPrdFrame[0]}
  [166] = {x=-81.661, y=89.19, z=14.348, rx=-171.233, ry=-11.16, rz=153, fatherId=fPrdFrame[0]}
  [167] = {x=-84.468, y=89.185, z=14.952, rx=-171.222, ry=-11.612, rz=153, fatherId=fPrdFrame[0]}
  [168] = {x=-87.274, y=89.18, z=15.581, rx=-171.21, ry=-12.066, rz=153, fatherId=fPrdFrame[0]}
  [169] = {x=-90.081, y=89.174, z=16.235, rx=-171.198, ry=-12.52, rz=153, fatherId=fPrdFrame[0]}
  [170] = {x=-92.887, y=89.169, z=16.913, rx=-171.185, ry=-12.974, rz=153, fatherId=fPrdFrame[0]}
  [171] = {x=-95.694, y=89.163, z=17.617, rx=-171.172, ry=-13.43, rz=153, fatherId=fPrdFrame[0]}
  [172] = {x=-98.5, y=89.157, z=18.346, rx=-171.158, ry=-13.886, rz=153, fatherId=fPrdFrame[0]}
  [173] = {x=-101.307, y=89.151, z=19.101, rx=-171.144, ry=-14.343, rz=153, fatherId=fPrdFrame[0]}
  [174] = {x=-104.113, y=89.145, z=19.88, rx=-171.129, ry=-14.802, rz=153, fatherId=fPrdFrame[0]}
  [175] = {x=-106.92, y=89.138, z=20.686, rx=-171.114, ry=-15.261, rz=153, fatherId=fPrdFrame[0]}
  [176] = {x=-109.726, y=89.132, z=21.517, rx=-171.098, ry=-15.721, rz=153, fatherId=fPrdFrame[0]}
  [177] = {x=-112.533, y=89.124, z=22.375, rx=-171.082, ry=-16.182, rz=153, fatherId=fPrdFrame[0]}
  [178] = {x=-115.339, y=89.117, z=23.259, rx=-171.065, ry=-16.644, rz=153, fatherId=fPrdFrame[0]}
  [179] = {x=-118.146, y=89.11, z=24.169, rx=-171.047, ry=-17.108, rz=153, fatherId=fPrdFrame[0]}
  [180] = {x=-120.952, y=89.102, z=25.105, rx=-171.029, ry=-17.572, rz=153, fatherId=fPrdFrame[0]}
  [181] = {x=-120.945, y=91.976, z=25.587, rx=-170.737, ry=-17.59, rz=153, fatherId=fPrdFrame[0]}
  [182] = {x=-118.139, y=91.984, z=24.649, rx=-170.756, ry=-17.125, rz=153, fatherId=fPrdFrame[0]}
  [183] = {x=-115.332, y=91.992, z=23.738, rx=-170.774, ry=-16.661, rz=153, fatherId=fPrdFrame[0]}
  [184] = {x=-112.526, y=91.999, z=22.854, rx=-170.792, ry=-16.198, rz=153, fatherId=fPrdFrame[0]}
  [185] = {x=-109.72, y=92.007, z=21.995, rx=-170.809, ry=-15.737, rz=153, fatherId=fPrdFrame[0]}
  [186] = {x=-106.913, y=92.014, z=21.163, rx=-170.825, ry=-15.276, rz=153, fatherId=fPrdFrame[0]}
  [187] = {x=-104.107, y=92.021, z=20.356, rx=-170.841, ry=-14.816, rz=153, fatherId=fPrdFrame[0]}
  [188] = {x=-101.301, y=92.027, z=19.576, rx=-170.856, ry=-14.358, rz=153, fatherId=fPrdFrame[0]}
  [189] = {x=-98.494, y=92.033, z=18.821, rx=-170.871, ry=-13.9, rz=153, fatherId=fPrdFrame[0]}
  [190] = {x=-95.688, y=92.04, z=18.091, rx=-170.885, ry=-13.443, rz=153, fatherId=fPrdFrame[0]}
  [191] = {x=-92.882, y=92.045, z=17.386, rx=-170.899, ry=-12.987, rz=153, fatherId=fPrdFrame[0]}
  [192] = {x=-90.075, y=92.051, z=16.707, rx=-170.912, ry=-12.532, rz=153, fatherId=fPrdFrame[0]}
  [193] = {x=-87.269, y=92.056, z=16.053, rx=-170.924, ry=-12.077, rz=153, fatherId=fPrdFrame[0]}
  [194] = {x=-84.463, y=92.062, z=15.423, rx=-170.936, ry=-11.624, rz=153, fatherId=fPrdFrame[0]}
  [195] = {x=-81.657, y=92.067, z=14.818, rx=-170.948, ry=-11.171, rz=153, fatherId=fPrdFrame[0]}
  [196] = {x=-78.85, y=92.071, z=14.238, rx=-170.959, ry=-10.719, rz=153, fatherId=fPrdFrame[0]}
  [197] = {x=-76.044, y=92.076, z=13.683, rx=-170.969, ry=-10.267, rz=153, fatherId=fPrdFrame[0]}
  [198] = {x=-73.238, y=92.08, z=13.151, rx=-170.979, ry=-9.816, rz=153, fatherId=fPrdFrame[0]}
  [199] = {x=-70.431, y=92.084, z=12.644, rx=-170.989, ry=-9.366, rz=153, fatherId=fPrdFrame[0]}
  [200] = {x=-67.625, y=92.088, z=12.162, rx=-170.998, ry=-8.916, rz=153, fatherId=fPrdFrame[0]}
  [201] = {x=-64.819, y=92.092, z=11.703, rx=-171.007, ry=-8.467, rz=153, fatherId=fPrdFrame[0]}
  [202] = {x=-62.013, y=92.096, z=11.268, rx=-171.015, ry=-8.019, rz=153, fatherId=fPrdFrame[0]}
  [203] = {x=-59.206, y=92.099, z=10.858, rx=-171.023, ry=-7.571, rz=153, fatherId=fPrdFrame[0]}
  [204] = {x=-56.4, y=92.102, z=10.471, rx=-171.03, ry=-7.123, rz=153, fatherId=fPrdFrame[0]}
  [205] = {x=-53.594, y=92.105, z=10.108, rx=-171.037, ry=-6.676, rz=153, fatherId=fPrdFrame[0]}
  [206] = {x=-50.788, y=92.108, z=9.769, rx=-171.043, ry=-6.229, rz=153, fatherId=fPrdFrame[0]}
  [207] = {x=-47.981, y=92.11, z=9.453, rx=-171.049, ry=-5.782, rz=153, fatherId=fPrdFrame[0]}
  [208] = {x=-45.175, y=92.113, z=9.161, rx=-171.054, ry=-5.336, rz=153, fatherId=fPrdFrame[0]}
  [209] = {x=-42.369, y=92.115, z=8.893, rx=-171.059, ry=-4.89, rz=153, fatherId=fPrdFrame[0]}
  [210] = {x=-39.563, y=92.117, z=8.648, rx=-171.064, ry=-4.445, rz=153, fatherId=fPrdFrame[0]}
  [211] = {x=-36.756, y=92.118, z=8.426, rx=-171.068, ry=-4, rz=153, fatherId=fPrdFrame[0]}
  [212] = {x=-33.95, y=92.12, z=8.228, rx=-171.072, ry=-3.555, rz=153, fatherId=fPrdFrame[0]}
  [213] = {x=-31.144, y=92.121, z=8.053, rx=-171.075, ry=-3.11, rz=153, fatherId=fPrdFrame[0]}
  [214] = {x=-28.338, y=92.123, z=7.902, rx=-171.078, ry=-2.665, rz=153, fatherId=fPrdFrame[0]}
  [215] = {x=-25.531, y=92.124, z=7.774, rx=-171.08, ry=-2.221, rz=153, fatherId=fPrdFrame[0]}
  [216] = {x=-22.725, y=92.124, z=7.67, rx=-171.082, ry=-1.776, rz=153, fatherId=fPrdFrame[0]}
  [217] = {x=-19.919, y=92.125, z=7.588, rx=-171.083, ry=-1.332, rz=153, fatherId=fPrdFrame[0]}
  [218] = {x=-17.112, y=92.126, z=7.53, rx=-171.084, ry=-0.888, rz=153, fatherId=fPrdFrame[0]}
  [219] = {x=-14.306, y=92.126, z=7.495, rx=-171.085, ry=-0.444, rz=153, fatherId=fPrdFrame[0]}
  [220] = {x=-11.5, y=92.126, z=7.483, rx=-171.085, rz=153, fatherId=fPrdFrame[0]}
  [221] = {x=-8.694, y=92.126, z=7.495, rx=-171.085, ry=0.444, rz=153, fatherId=fPrdFrame[0]}
  [222] = {x=-5.888, y=92.126, z=7.53, rx=-171.084, ry=0.888, rz=153, fatherId=fPrdFrame[0]}
  [223] = {x=-3.081, y=92.125, z=7.588, rx=-171.083, ry=1.332, rz=153, fatherId=fPrdFrame[0]}
  [224] = {x=-0.275, y=92.124, z=7.67, rx=-171.082, ry=1.776, rz=153, fatherId=fPrdFrame[0]}
  [225] = {x=2.531, y=92.124, z=7.774, rx=-171.08, ry=2.221, rz=153, fatherId=fPrdFrame[0]}
  [226] = {x=5.338, y=92.123, z=7.902, rx=-171.078, ry=2.665, rz=153, fatherId=fPrdFrame[0]}
  [227] = {x=8.144, y=92.121, z=8.053, rx=-171.075, ry=3.11, rz=153, fatherId=fPrdFrame[0]}
  [228] = {x=10.95, y=92.12, z=8.228, rx=-171.072, ry=3.555, rz=153, fatherId=fPrdFrame[0]}
  [229] = {x=13.756, y=92.118, z=8.426, rx=-171.068, ry=4, rz=153, fatherId=fPrdFrame[0]}
  [230] = {x=16.563, y=92.117, z=8.648, rx=-171.064, ry=4.445, rz=153, fatherId=fPrdFrame[0]}
  [231] = {x=19.369, y=92.115, z=8.893, rx=-171.059, ry=4.89, rz=153, fatherId=fPrdFrame[0]}
  [232] = {x=22.175, y=92.113, z=9.161, rx=-171.054, ry=5.336, rz=153, fatherId=fPrdFrame[0]}
  [233] = {x=24.981, y=92.11, z=9.453, rx=-171.049, ry=5.782, rz=153, fatherId=fPrdFrame[0]}
  [234] = {x=27.788, y=92.108, z=9.769, rx=-171.043, ry=6.229, rz=153, fatherId=fPrdFrame[0]}
  [235] = {x=30.594, y=92.105, z=10.108, rx=-171.037, ry=6.676, rz=153, fatherId=fPrdFrame[0]}
  [236] = {x=33.4, y=92.102, z=10.471, rx=-171.03, ry=7.123, rz=153, fatherId=fPrdFrame[0]}
  [237] = {x=36.206, y=92.099, z=10.858, rx=-171.023, ry=7.571, rz=153, fatherId=fPrdFrame[0]}
  [238] = {x=39.013, y=92.096, z=11.268, rx=-171.015, ry=8.019, rz=153, fatherId=fPrdFrame[0]}
  [239] = {x=41.819, y=92.092, z=11.703, rx=-171.007, ry=8.467, rz=153, fatherId=fPrdFrame[0]}
  [240] = {x=44.625, y=92.088, z=12.162, rx=-170.998, ry=8.916, rz=153, fatherId=fPrdFrame[0]}
  [241] = {x=47.431, y=92.084, z=12.644, rx=-170.989, ry=9.366, rz=153, fatherId=fPrdFrame[0]}
  [242] = {x=50.238, y=92.08, z=13.151, rx=-170.979, ry=9.816, rz=153, fatherId=fPrdFrame[0]}
  [243] = {x=53.044, y=92.076, z=13.683, rx=-170.969, ry=10.267, rz=153, fatherId=fPrdFrame[0]}
  [244] = {x=55.85, y=92.071, z=14.238, rx=-170.959, ry=10.719, rz=153, fatherId=fPrdFrame[0]}
  [245] = {x=58.657, y=92.067, z=14.818, rx=-170.948, ry=11.171, rz=153, fatherId=fPrdFrame[0]}
  [246] = {x=61.463, y=92.062, z=15.423, rx=-170.936, ry=11.624, rz=153, fatherId=fPrdFrame[0]}
  [247] = {x=64.269, y=92.056, z=16.053, rx=-170.924, ry=12.077, rz=153, fatherId=fPrdFrame[0]}
